KUKA KRL program: EPS_2_25862_MH3A_A_20251016034258.src

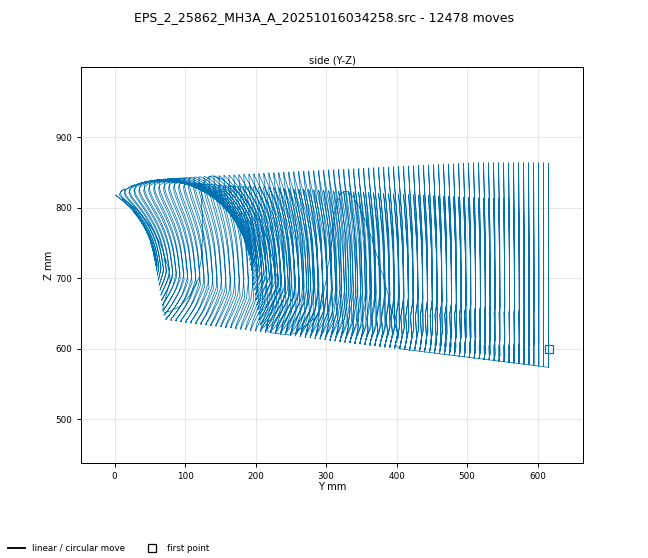
[picture p0: tool path of EPS_2_25862_MH3A_A_20251016034258.src, 12478 of 12480 moves have a stored position in this frame; points joined in program order, loops and branches not executed]
&ACCESS RVP
&REL 4
&COMMENT QRS 19112012
&PARAM EDITMASK = *
DEF PART()
EXT BAS (BAS_COMMAND :IN,REAL :IN )
INT I
BAS (#INITMOV,0 )

;KUKA QRS Post kuka4.cps  Date:22-06-2017 !

File_ID=2889

QRS_PRE_INIT()

;Init var - Until changes are made in qrs_pre_init
Outlet_Square_prg=0
Inlet_1_Square_prg=0
Inlet_2_Square_prg=0
Inlet_3_Square_prg=0
Inlet_4_Square_prg=0
Inlet_5_Square_prg=0

Outlet_1={X 0.000, Y 513.730, Z 763.500, B 0.000, E1 0.000 }
Inlet_1={X 0.000, Y 517.300, Z 713.500, B 0.000, E1 225.000 }
Outlet_1_type=201
Inlet_1_type=201
;QRS#1=Sidecore dimensions
;QRS#2=200-8" PVC SDR 35
;QRS#3=200-8" PVC SDR 35
;QRS#4=
;QRS#5=
;QRS#6=
;QRS#7=
;QRS#8=
;QRS#9=12-08 PSX
;QRS#10=12-08 PSX
;QRS#11=
;QRS#12=
;QRS#13=
;QRS#14=
;QRS#15=
;QRS#16=1220x127x1143 3,75'
;QRS#17=EPS Height
;QRS#18=864
;QRS#19=*
;QRS#20= UPDATED VERSION 22-06-2017
;QRS#21=*
Outlet_Square=0100
Inlet_1_Square=0100
Inlet_2_Square=0
Inlet_3_Square=0
Inlet_4_Square=0
Inlet_5_Square=0
Mill_Square=1
Outlet_Square_Prg=204
Inlet_1_Square_prg=204

QRS_INIT()

$ADVANCE=5

; T1
PTP {E1 173.596,E2 173.596}
PTP {X 0,Y 615.504,A -85,B 0,C 180,E1 173.596,E2 173.596,E3 0,E4 0,E5 0,E6 0}
QRS_SPEED_INIT()
LIN {X 0,Y 615.504,Z 600,A -85,B 0,C 180,E1 173.596,E2 173.596,E3 0,E4 0,E5 0,E6 0} C_VEL
LIN {X 0,Y 615.504,Z 583.862,A -85,B 0,C 180,E1 173.596,E2 173.596} C_VEL
LIN {X 0,Y 615.504,Z 575.681,A -85,B 0,C 180,E1 173.596,E2 173.596} C_VEL
LIN {X 0,Y 615.487,Z 573.681,A -85,B 0,C 180,E1 173.41,E2 173.41} C_VEL
LIN {X 0,Y 615.476,Z 573.691,A -85,B 0,C 180,E1 170.801,E2 170.801} C_VEL
LIN {X 0,Y 615.486,Z 573.696,A -85,B 0,C 180,E1 168.14,E2 168.14} C_VEL
LIN {X 0,Y 615.48,Z 573.683,A -85,B 0,C 180,E1 165.451,E2 165.451} C_VEL
LIN {X 0,Y 615.477,Z 573.689,A -85,B 0,C 180,E1 162.73,E2 162.73} C_VEL
LIN {X 0,Y 615.485,Z 573.695,A -85,B 0,C 180,E1 159.968,E2 159.968} C_VEL
LIN {X 0,Y 615.486,Z 573.681,A -85,B 0,C 180,E1 157.156,E2 157.156} C_VEL
LIN {X 0,Y 615.485,Z 573.696,A -85,B 0,C 180,E1 154.285,E2 154.285} C_VEL
LIN {X 0,Y 615.476,Z 573.69,A -85,B 0,C 180,E1 151.549,E2 151.549} C_VEL
LIN {X 0,Y 615.483,Z 573.682,A -85,B 0,C 180,E1 148.912,E2 148.912} C_VEL
LIN {X 0,Y 615.495,Z 573.699,A -85,B 0,C 180,E1 145.979,E2 145.979} C_VEL
LIN {X 0,Y 615.486,Z 573.682,A -85,B 0,C 180,E1 143.062,E2 143.062} C_VEL
LIN {X 0,Y 615.477,Z 573.691,A -85,B 0,C 180,E1 140.25,E2 140.25} C_VEL
LIN {X 0,Y 615.489,Z 573.697,A -85,B 0,C 180,E1 137.648,E2 137.648} C_VEL
LIN {X 0,Y 615.48,Z 573.684,A -85,B 0,C 180,E1 134.931,E2 134.931} C_VEL
LIN {X 0,Y 615.477,Z 573.691,A -85,B 0,C 180,E1 132.08,E2 132.08} C_VEL
LIN {X 0,Y 615.493,Z 573.697,A -85,B 0,C 180,E1 129.749,E2 129.749} C_VEL
LIN {X 0,Y 615.48,Z 573.685,A -85,B 0,C 180,E1 126.936,E2 126.936} C_VEL
LIN {X 0,Y 615.49,Z 573.681,A -85,B 0,C 180,E1 124.702,E2 124.702} C_VEL
LIN {X 0,Y 615.484,Z 573.682,A -85,B 0,C 180,E1 122.331,E2 122.331} C_VEL
LIN {X 0,Y 615.494,Z 573.7,A -85,B 0,C 180,E1 119.405,E2 119.405} C_VEL
LIN {X 0,Y 615.491,Z 573.68,A -85,B 0,C 180,E1 116.443,E2 116.443} C_VEL
LIN {X 0,Y 615.487,Z 573.695,A -85,B 0,C 180,E1 113.556,E2 113.556} C_VEL
LIN {X 0,Y 615.479,Z 573.687,A -85,B 0,C 180,E1 110.73,E2 110.73} C_VEL
LIN {X 0,Y 615.478,Z 573.685,A -85,B 0,C 180,E1 107.957,E2 107.957} C_VEL
LIN {X 0,Y 615.492,Z 573.701,A -85,B 0,C 180,E1 105.226,E2 105.226} C_VEL
LIN {X 0,Y 615.479,Z 573.686,A -85,B 0,C 180,E1 102.53,E2 102.53} C_VEL
LIN {X 0,Y 615.48,Z 573.684,A -85,B 0,C 180,E1 99.862,E2 99.862} C_VEL
LIN {X 0,Y 615.489,Z 573.696,A -85,B 0,C 180,E1 97.215,E2 97.215} C_VEL
LIN {X 0,Y 615.48,Z 573.69,A -85,B 0,C 180,E1 94.584,E2 94.584} C_VEL
LIN {X 0,Y 615.493,Z 573.68,A -85,B 0,C 180,E1 91.963,E2 91.963} C_VEL
LIN {X 0,Y 615.474,Z 573.691,A -85,B 0,C 180,E1 89.346,E2 89.346} C_VEL
LIN {X 0,Y 615.49,Z 573.697,A -85,B 0,C 180,E1 86.727,E2 86.727} C_VEL
LIN {X 0,Y 615.486,Z 573.683,A -85,B 0,C 180,E1 84.102,E2 84.102} C_VEL
LIN {X 0,Y 615.477,Z 573.685,A -85,B 0,C 180,E1 81.463,E2 81.463} C_VEL
LIN {X 0,Y 615.498,Z 573.697,A -85,B 0,C 180,E1 78.807,E2 78.807} C_VEL
LIN {X 0,Y 615.483,Z 573.686,A -85,B 0,C 180,E1 76.067,E2 76.067} C_VEL
LIN {X 0,Y 615.478,Z 573.684,A -85,B 0,C 180,E1 73.414,E2 73.414} C_VEL
LIN {X 0,Y 615.489,Z 573.699,A -85,B 0,C 180,E1 70.663,E2 70.663} C_VEL
LIN {X 0,Y 615.491,Z 573.681,A -85,B 0,C 180,E1 67.652,E2 67.652} C_VEL
LIN {X 0,Y 615.475,Z 573.688,A -85,B 0,C 180,E1 65.008,E2 65.008} C_VEL
LIN {X 0,Y 615.477,Z 573.878,A -85,B 0,C 180,E1 62.956,E2 62.956} C_VEL
LIN {X 0,Y 615.476,Z 589.581,A -85,B 0,C 180,E1 60.206,E2 60.206} C_VEL
LIN {X 0,Y 615.478,Z 603.411,A -85,B 0,C 180,E1 57.811,E2 57.811} C_VEL
LIN {X 0,Y 615.492,Z 710.1,A -85,B 0,C 180,E1 56.539,E2 56.539} C_VEL
LIN {X 0,Y 615.486,Z 723.119,A -85,B 0,C 180,E1 56.252,E2 56.252} C_VEL
LIN {X 0,Y 615.483,Z 735.365,A -85,B 0,C 180,E1 55.851,E2 55.851} C_VEL
LIN {X 0,Y 615.489,Z 747.801,A -85,B 0,C 180,E1 55.298,E2 55.298} C_VEL
LIN {X 0,Y 615.478,Z 758.469,A -85,B 0,C 180,E1 54.686,E2 54.686} C_VEL
LIN {X 0,Y 615.5,Z 769.773,A -85,B 0,C 180,E1 53.871,E2 53.871} C_VEL
LIN {X 0,Y 615.497,Z 778.829,A -85,B 0,C 180,E1 53.062,E2 53.062} C_VEL
LIN {X 0,Y 615.494,Z 786.885,A -85,B 0,C 180,E1 52.18,E2 52.18} C_VEL
LIN {X 0,Y 615.493,Z 794.893,A -85,B 0,C 180,E1 51.097,E2 51.097} C_VEL
LIN {X 0,Y 615.498,Z 799.899,A -85,B 0,C 180,E1 50.252,E2 50.252} C_VEL
LIN {X 0,Y 615.498,Z 805.113,A -85,B 0,C 180,E1 49.15,E2 49.15} C_VEL
LIN {X 0,Y 615.498,Z 809.309,A -85,B 0,C 180,E1 47.918,E2 47.918} C_VEL
LIN {X 0,Y 615.496,Z 811.875,A -85,B 0,C 180,E1 46.757,E2 46.757} C_VEL
LIN {X 0,Y 615.495,Z 813.002,A -85,B 0,C 180,E1 45.853,E2 45.853} C_VEL
LIN {X 0,Y 615.495,Z 813.388,A -85,B 0,C 180,E1 44.934,E2 44.934} C_VEL
LIN {X 0,Y 615.493,Z 812.962,A -85,B 0,C 180,E1 44,E2 44} C_VEL
LIN {X 0,Y 615.497,Z 811.704,A -85,B 0,C 180,E1 43.05,E2 43.05} C_VEL
LIN {X 0,Y 615.496,Z 809.552,A -85,B 0,C 180,E1 42.083,E2 42.083} C_VEL
LIN {X 0,Y 615.493,Z 806.404,A -85,B 0,C 180,E1 41.097,E2 41.097} C_VEL
LIN {X 0,Y 615.497,Z 802.114,A -85,B 0,C 180,E1 40.092,E2 40.092} C_VEL
LIN {X 0,Y 615.497,Z 796.474,A -85,B 0,C 180,E1 39.065,E2 39.065} C_VEL
LIN {X 0,Y 615.495,Z 789.205,A -85,B 0,C 180,E1 38.015,E2 38.015} C_VEL
LIN {X 0,Y 615.498,Z 781.195,A -85,B 0,C 180,E1 37.09,E2 37.09} C_VEL
LIN {X 0,Y 615.499,Z 772.601,A -85,B 0,C 180,E1 36.276,E2 36.276} C_VEL
LIN {X 0,Y 615.495,Z 762.802,A -85,B 0,C 180,E1 35.514,E2 35.514} C_VEL
LIN {X 0,Y 615.483,Z 751.624,A -85,B 0,C 180,E1 34.815,E2 34.815} C_VEL
LIN {X 0,Y 615.489,Z 739.667,A -85,B 0,C 180,E1 34.233,E2 34.233} C_VEL
LIN {X 0,Y 615.48,Z 727.257,A -85,B 0,C 180,E1 33.778,E2 33.778} C_VEL
LIN {X 0,Y 615.474,Z 714.959,A -85,B 0,C 180,E1 33.46,E2 33.46} C_VEL
LIN {X 0,Y 615.48,Z 700.03,A -85,B 0,C 180,E1 33.236,E2 33.236} C_VEL
LIN {X 0,Y 615.483,Z 603.35,A -85,B 0,C 180,E1 32.089,E2 32.089} C_VEL
LIN {X 0,Y 615.49,Z 586.786,A -85,B 0,C 180,E1 29.218,E2 29.218} C_VEL
LIN {X 0,Y 615.496,Z 573.683,A -85,B 0,C 180,E1 26.897,E2 26.897} C_VEL
LIN {X 0,Y 615.485,Z 573.686,A -85,B 0,C 180,E1 24.011,E2 24.011} C_VEL
LIN {X 0,Y 615.495,Z 573.7,A -85,B 0,C 180,E1 21.431,E2 21.431} C_VEL
LIN {X 0,Y 615.483,Z 573.683,A -85,B 0,C 180,E1 18.608,E2 18.608} C_VEL
LIN {X 0,Y 615.483,Z 573.686,A -85,B 0,C 180,E1 15.905,E2 15.905} C_VEL
LIN {X 0,Y 615.495,Z 573.697,A -85,B 0,C 180,E1 13.201,E2 13.201} C_VEL
LIN {X 0,Y 615.485,Z 573.683,A -85,B 0,C 180,E1 10.527,E2 10.527} C_VEL
LIN {X 0,Y 615.482,Z 573.685,A -85,B 0,C 180,E1 7.875,E2 7.875} C_VEL
LIN {X 0,Y 615.487,Z 573.701,A -85,B 0,C 180,E1 5.241,E2 5.241} C_VEL
LIN {X 0,Y 615.496,Z 573.684,A -85,B 0,C 180,E1 2.617,E2 2.617} C_VEL
LIN {X 0,Y 615.476,Z 573.684,A -85,B 0,C 180,E1 0,E2 0} C_VEL
LIN {X 0,Y 615.496,Z 573.69,A -85,B 0,C 180,E1 -2.618,E2 -2.618} C_VEL
LIN {X 0,Y 615.49,Z 573.691,A -85,B 0,C 180,E1 -5.242,E2 -5.242} C_VEL
LIN {X 0,Y 615.482,Z 573.683,A -85,B 0,C 180,E1 -7.876,E2 -7.876} C_VEL
LIN {X 0,Y 615.484,Z 573.688,A -85,B 0,C 180,E1 -10.527,E2 -10.527} C_VEL
LIN {X 0,Y 615.49,Z 573.696,A -85,B 0,C 180,E1 -13.201,E2 -13.201} C_VEL
LIN {X 0,Y 615.483,Z 573.683,A -85,B 0,C 180,E1 -15.906,E2 -15.906} C_VEL
LIN {X 0,Y 615.484,Z 573.688,A -85,B 0,C 180,E1 -18.646,E2 -18.646} C_VEL
LIN {X 0,Y 615.486,Z 573.693,A -85,B 0,C 180,E1 -21.432,E2 -21.432} C_VEL
LIN {X 0,Y 615.478,Z 573.684,A -85,B 0,C 180,E1 -24.273,E2 -24.273} C_VEL
LIN {X 0,Y 615.492,Z 573.695,A -85,B 0,C 180,E1 -27.049,E2 -27.049} C_VEL
LIN {X 0,Y 615.49,Z 573.685,A -85,B 0,C 180,E1 -29.797,E2 -29.797} C_VEL
LIN {X 0,Y 615.477,Z 573.684,A -85,B 0,C 180,E1 -32.458,E2 -32.458} C_VEL
LIN {X 0,Y 615.477,Z 573.689,A -85,B 0,C 180,E1 -34.816,E2 -34.816} C_VEL
LIN {X 0,Y 615.492,Z 573.697,A -85,B 0,C 180,E1 -37.242,E2 -37.242} C_VEL
LIN {X 0,Y 615.495,Z 573.682,A -85,B 0,C 180,E1 -40.092,E2 -40.092} C_VEL
LIN {X 0,Y 615.488,Z 573.681,A -85,B 0,C 180,E1 -42.353,E2 -42.353} C_VEL
LIN {X 0,Y 615.481,Z 573.691,A -85,B 0,C 180,E1 -45.07,E2 -45.07} C_VEL
LIN {X 0,Y 615.483,Z 573.69,A -85,B 0,C 180,E1 -47.921,E2 -47.921} C_VEL
LIN {X 0,Y 615.494,Z 573.681,A -85,B 0,C 180,E1 -50.252,E2 -50.252} C_VEL
LIN {X 0,Y 615.478,Z 573.689,A -85,B 0,C 180,E1 -53.065,E2 -53.065} C_VEL
LIN {X 0,Y 615.49,Z 573.691,A -85,B 0,C 180,E1 -55.3,E2 -55.3} C_VEL
LIN {X 0,Y 615.494,Z 573.7,A -85,B 0,C 180,E1 -57.669,E2 -57.669} C_VEL
LIN {X 0,Y 615.493,Z 573.68,A -85,B 0,C 180,E1 -60.595,E2 -60.595} C_VEL
LIN {X 0,Y 615.491,Z 573.696,A -85,B 0,C 180,E1 -63.557,E2 -63.557} C_VEL
LIN {X 0,Y 615.489,Z 573.683,A -85,B 0,C 180,E1 -66.444,E2 -66.444} C_VEL
LIN {X 0,Y 615.475,Z 573.827,A -85,B 0,C 180,E1 -67.067,E2 -67.067} C_VEL
LIN {X 0,Y 615.486,Z 594.759,A -85,B 0,C 180,E1 -69.837,E2 -69.837} C_VEL
LIN {X 0,Y 615.497,Z 616.999,A -85,B 0,C 180,E1 -72.73,E2 -72.73} C_VEL
LIN {X 0,Y 615.484,Z 639.434,A -85,B 0,C 180,E1 -75.606,E2 -75.606} C_VEL
LIN {X 0,Y 615.478,Z 651.3,A -85,B 0,C 180,E1 -77.114,E2 -77.114} C_VEL
LIN {X 0,Y 615.477,Z 759.849,A -85,B 0,C 180,E1 -78.411,E2 -78.411} C_VEL
LIN {X 0,Y 615.488,Z 772.354,A -85,B 0,C 180,E1 -78.682,E2 -78.682} C_VEL
LIN {X 0,Y 615.496,Z 785.512,A -85,B 0,C 180,E1 -79.109,E2 -79.109} C_VEL
LIN {X 0,Y 615.484,Z 797.482,A -85,B 0,C 180,E1 -79.64,E2 -79.64} C_VEL
LIN {X 0,Y 615.483,Z 809,A -85,B 0,C 180,E1 -80.304,E2 -80.304} C_VEL
LIN {X 0,Y 615.499,Z 819.344,A -85,B 0,C 180,E1 -81.05,E2 -81.05} C_VEL
LIN {X 0,Y 615.497,Z 827.814,A -85,B 0,C 180,E1 -81.794,E2 -81.794} C_VEL
LIN {X 0,Y 615.498,Z 835.608,A -85,B 0,C 180,E1 -82.62,E2 -82.62} C_VEL
LIN {X 0,Y 615.496,Z 843.204,A -85,B 0,C 180,E1 -83.608,E2 -83.608} C_VEL
LIN {X 0,Y 615.498,Z 850.205,A -85,B 0,C 180,E1 -84.759,E2 -84.759} C_VEL
LIN {X 0,Y 615.494,Z 854.852,A -85,B 0,C 180,E1 -85.744,E2 -85.744} C_VEL
LIN {X 0,Y 615.496,Z 858.399,A -85,B 0,C 180,E1 -86.727,E2 -86.727} C_VEL
LIN {X 0,Y 615.497,Z 860.233,A -85,B 0,C 180,E1 -87.382,E2 -87.382} C_VEL
LIN {X 0,Y 615.496,Z 861.608,A -85,B 0,C 180,E1 -88.037,E2 -88.037} C_VEL
LIN {X 0,Y 615.496,Z 863.174,A -85,B 0,C 180,E1 -89.346,E2 -89.346} C_VEL
LIN {X 0,Y 615.494,Z 863.389,A -85,B 0,C 180,E1 -90,E2 -90} C_VEL
LIN {X 0,Y 615.496,Z 862.58,A -85,B 0,C 180,E1 -91.309,E2 -91.309} C_VEL
LIN {X 0,Y 615.496,Z 861.608,A -85,B 0,C 180,E1 -91.963,E2 -91.963} C_VEL
LIN {X 0,Y 615.497,Z 860.233,A -85,B 0,C 180,E1 -92.618,E2 -92.618} C_VEL
LIN {X 0,Y 615.496,Z 857.35,A -85,B 0,C 180,E1 -93.601,E2 -93.601} C_VEL
LIN {X 0,Y 615.498,Z 853.442,A -85,B 0,C 180,E1 -94.584,E2 -94.584} C_VEL
LIN {X 0,Y 615.499,Z 848.406,A -85,B 0,C 180,E1 -95.57,E2 -95.57} C_VEL
LIN {X 0,Y 615.497,Z 841.87,A -85,B 0,C 180,E1 -96.583,E2 -96.583} C_VEL
LIN {X 0,Y 615.497,Z 834.135,A -85,B 0,C 180,E1 -97.545,E2 -97.545} C_VEL
LIN {X 0,Y 615.498,Z 826.047,A -85,B 0,C 180,E1 -98.371,E2 -98.371} C_VEL
LIN {X 0,Y 615.499,Z 816.17,A -85,B 0,C 180,E1 -99.198,E2 -99.198} C_VEL
LIN {X 0,Y 615.487,Z 804.986,A -85,B 0,C 180,E1 -99.945,E2 -99.945} C_VEL
LIN {X 0,Y 615.483,Z 794.029,A -85,B 0,C 180,E1 -100.527,E2 -100.527} C_VEL
LIN {X 0,Y 615.496,Z 781.436,A -85,B 0,C 180,E1 -101.042,E2 -101.042} C_VEL
LIN {X 0,Y 615.483,Z 769.078,A -85,B 0,C 180,E1 -101.401,E2 -101.401} C_VEL
LIN {X 0,Y 615.477,Z 755.49,A -85,B 0,C 180,E1 -101.652,E2 -101.652} C_VEL
LIN {X 0,Y 615.478,Z 651.3,A -85,B 0,C 180,E1 -102.886,E2 -102.886} C_VEL
LIN {X 0,Y 615.48,Z 630.263,A -85,B 0,C 180,E1 -105.565,E2 -105.565} C_VEL
LIN {X 0,Y 615.498,Z 609.208,A -85,B 0,C 180,E1 -108.278,E2 -108.278} C_VEL
LIN {X 0,Y 615.489,Z 586.457,A -85,B 0,C 180,E1 -111.256,E2 -111.256} C_VEL
LIN {X 0,Y 615.477,Z 573.685,A -85,B 0,C 180,E1 -112.978,E2 -112.978} C_VEL
LIN {X 0,Y 615.484,Z 573.686,A -85,B 0,C 180,E1 -115.715,E2 -115.715} C_VEL
LIN {X 0,Y 615.494,Z 573.697,A -85,B 0,C 180,E1 -118.451,E2 -118.451} C_VEL
LIN {X 0,Y 615.473,Z 573.686,A -85,B 0,C 180,E1 -121.083,E2 -121.083} C_VEL
LIN {X 0,Y 615.495,Z 573.679,A -85,B 0,C 180,E1 -123.535,E2 -123.535} C_VEL
LIN {X 0,Y 615.487,Z 573.7,A -85,B 0,C 180,E1 -126.424,E2 -126.424} C_VEL
LIN {X 0,Y 615.476,Z 573.689,A -85,B 0,C 180,E1 -129.06,E2 -129.06} C_VEL
LIN {X 0,Y 615.481,Z 573.683,A -85,B 0,C 180,E1 -131.473,E2 -131.473} C_VEL
LIN {X 0,Y 615.481,Z 573.688,A -85,B 0,C 180,E1 -134.149,E2 -134.149} C_VEL
LIN {X 0,Y 615.484,Z 573.693,A -85,B 0,C 180,E1 -136.951,E2 -136.951} C_VEL
LIN {X 0,Y 615.473,Z 573.687,A -85,B 0,C 180,E1 -139.392,E2 -139.392} C_VEL
LIN {X 0,Y 615.486,Z 573.682,A -85,B 0,C 180,E1 -141.986,E2 -141.986} C_VEL
LIN {X 0,Y 615.48,Z 573.69,A -85,B 0,C 180,E1 -144.383,E2 -144.383} C_VEL
LIN {X 0,Y 615.486,Z 573.699,A -85,B 0,C 180,E1 -146.763,E2 -146.763} C_VEL
LIN {X 0,Y 615.487,Z 573.696,A -85,B 0,C 180,E1 -149.08,E2 -149.08} C_VEL
LIN {X 0,Y 615.476,Z 573.687,A -85,B 0,C 180,E1 -151.549,E2 -151.549} C_VEL
LIN {X 0,Y 615.486,Z 573.683,A -85,B 0,C 180,E1 -154.284,E2 -154.284} C_VEL
LIN {X 0,Y 615.488,Z 573.698,A -85,B 0,C 180,E1 -157.155,E2 -157.155} C_VEL
LIN {X 0,Y 615.485,Z 573.682,A -85,B 0,C 180,E1 -159.967,E2 -159.967} C_VEL
LIN {X 0,Y 615.479,Z 573.69,A -85,B 0,C 180,E1 -162.729,E2 -162.729} C_VEL
LIN {X 0,Y 615.48,Z 573.695,A -85,B 0,C 180,E1 -165.45,E2 -165.45} C_VEL
LIN {X 0,Y 615.485,Z 573.682,A -85,B 0,C 180,E1 -168.139,E2 -168.139} C_VEL
LIN {X 0,Y 615.478,Z 573.689,A -85,B 0,C 180,E1 -170.801,E2 -170.801} C_VEL
LIN {X 0,Y 615.489,Z 573.698,A -85,B 0,C 180,E1 -173.443,E2 -173.443} C_VEL
LIN {X 0,Y 615.477,Z 573.685,A -85,B 0,C 180,E1 -176.071,E2 -176.071} C_VEL
LIN {X 0,Y 615.485,Z 573.683,A -85,B 0,C 180,E1 -178.691,E2 -178.691} C_VEL
LIN {X 0,Y 615.487,Z 573.696,A -85,B 0,C 180,E1 -181.308,E2 -181.308} C_VEL
LIN {X 0,Y 615.477,Z 573.691,A -85,B 0,C 180,E1 -183.928,E2 -183.928} C_VEL
LIN {X 0,Y 615.487,Z 573.681,A -85,B 0,C 180,E1 -186.59,E2 -186.59} C_VEL
LIN {X 0,Y 614.805,Z 573.839,A -85,B 0,C 180,E1 -187.136,E2 -187.136} C_VEL
LIN {X 0,Y 611.964,Z 574.253,A -85,B 0,C 180,E1 -188.022,E2 -188.022} C_VEL
LIN {X 0,Y 609.571,Z 574.564,A -85,B 0,C 180,E1 -188.735,E2 -188.735} C_VEL
LIN {X 0,Y 608.539,Z 574.682,A -85,B 0,C 180,E1 -189.284,E2 -189.284} C_VEL
LIN {X 0,Y 608.452,Z 574.691,A -85,B 0,C 180,E1 -189.47,E2 -189.47} C_VEL
LIN {X 0,Y 608.46,Z 574.691,A -85,B 0,C 180,E1 -191.999,E2 -191.999} C_VEL
LIN {X 0,Y 608.467,Z 574.685,A -85,B 0,C 180,E1 -194.72,E2 -194.72} C_VEL
LIN {X 0,Y 608.446,Z 574.693,A -85,B 0,C 180,E1 -197.476,E2 -197.476} C_VEL
LIN {X 0,Y 608.459,Z 574.689,A -85,B 0,C 180,E1 -200.274,E2 -200.274} C_VEL
LIN {X 0,Y 608.447,Z 574.688,A -85,B 0,C 180,E1 -203.124,E2 -203.124} C_VEL
LIN {X 0,Y 608.466,Z 574.693,A -85,B 0,C 180,E1 -205.723,E2 -205.723} C_VEL
LIN {X 0,Y 608.444,Z 574.693,A -85,B 0,C 180,E1 -208.267,E2 -208.267} C_VEL
LIN {X 0,Y 608.47,Z 574.687,A -85,B 0,C 180,E1 -210.544,E2 -210.544} C_VEL
LIN {X 0,Y 608.45,Z 574.687,A -85,B 0,C 180,E1 -212.879,E2 -212.879} C_VEL
LIN {X 0,Y 608.434,Z 574.689,A -85,B 0,C 180,E1 -215.278,E2 -215.278} C_VEL
LIN {X 0,Y 608.471,Z 574.689,A -85,B 0,C 180,E1 -217.746,E2 -217.746} C_VEL
LIN {X 0,Y 608.472,Z 574.693,A -85,B 0,C 180,E1 -220.333,E2 -220.333} C_VEL
LIN {X 0,Y 608.483,Z 574.683,A -85,B 0,C 180,E1 -223.312,E2 -223.312} C_VEL
LIN {X 0,Y 608.465,Z 574.693,A -85,B 0,C 180,E1 -226.132,E2 -226.132} C_VEL
LIN {X 0,Y 608.447,Z 574.69,A -85,B 0,C 180,E1 -228.824,E2 -228.824} C_VEL
LIN {X 0,Y 608.462,Z 574.685,A -85,B 0,C 180,E1 -231.413,E2 -231.413} C_VEL
LIN {X 0,Y 608.471,Z 574.687,A -85,B 0,C 180,E1 -233.951,E2 -233.951} C_VEL
LIN {X 0,Y 608.467,Z 574.694,A -85,B 0,C 180,E1 -236.33,E2 -236.33} C_VEL
LIN {X 0,Y 608.471,Z 574.692,A -85,B 0,C 180,E1 -238.728,E2 -238.728} C_VEL
LIN {X 0,Y 608.473,Z 574.684,A -85,B 0,C 180,E1 -241.379,E2 -241.379} C_VEL
LIN {X 0,Y 608.443,Z 574.689,A -85,B 0,C 180,E1 -243.965,E2 -243.965} C_VEL
LIN {X 0,Y 608.461,Z 574.688,A -85,B 0,C 180,E1 -246.156,E2 -246.156} C_VEL
LIN {X 0,Y 608.47,Z 574.689,A -85,B 0,C 180,E1 -248.309,E2 -248.309} C_VEL
LIN {X 0,Y 608.465,Z 574.688,A -85,B 0,C 180,E1 -251.284,E2 -251.284} C_VEL
LIN {X 0,Y 608.456,Z 574.686,A -85,B 0,C 180,E1 -253.906,E2 -253.906} C_VEL
LIN {X 0,Y 608.469,Z 574.692,A -85,B 0,C 180,E1 -256.644,E2 -256.644} C_VEL
LIN {X 0,Y 608.459,Z 574.689,A -85,B 0,C 180,E1 -259.35,E2 -259.35} C_VEL
LIN {X 0,Y 608.473,Z 574.684,A -85,B 0,C 180,E1 -262.033,E2 -262.033} C_VEL
LIN {X 0,Y 608.465,Z 574.691,A -85,B 0,C 180,E1 -264.698,E2 -264.698} C_VEL
LIN {X 0,Y 608.472,Z 574.69,A -85,B 0,C 180,E1 -267.352,E2 -267.352} C_VEL
LIN {X 0,Y 608.477,Z 574.684,A -85,B 0,C 180,E1 -270,E2 -270} C_VEL
LIN {X 0,Y 608.469,Z 574.688,A -85,B 0,C 180,E1 -272.648,E2 -272.648} C_VEL
LIN {X 0,Y 608.469,Z 574.694,A -85,B 0,C 180,E1 -275.302,E2 -275.302} C_VEL
LIN {X 0,Y 608.475,Z 574.685,A -85,B 0,C 180,E1 -277.967,E2 -277.967} C_VEL
LIN {X 0,Y 608.456,Z 574.688,A -85,B 0,C 180,E1 -280.65,E2 -280.65} C_VEL
LIN {X 0,Y 608.47,Z 574.695,A -85,B 0,C 180,E1 -283.356,E2 -283.356} C_VEL
LIN {X 0,Y 608.458,Z 574.687,A -85,B 0,C 180,E1 -286.093,E2 -286.093} C_VEL
LIN {X 0,Y 608.451,Z 574.689,A -85,B 0,C 180,E1 -288.869,E2 -288.869} C_VEL
LIN {X 0,Y 608.472,Z 574.691,A -85,B 0,C 180,E1 -291.691,E2 -291.691} C_VEL
LIN {X 0,Y 608.451,Z 574.687,A -85,B 0,C 180,E1 -294.571,E2 -294.571} C_VEL
LIN {X 0,Y 608.46,Z 574.713,A -85,B 0,C 180,E1 -296.963,E2 -296.963} C_VEL
LIN {X 0,Y 608.48,Z 589.567,A -85,B 0,C 180,E1 -299.588,E2 -299.588} C_VEL
LIN {X 0,Y 608.442,Z 603.672,A -85,B 0,C 180,E1 -302.046,E2 -302.046} C_VEL
LIN {X 0,Y 608.562,Z 710.327,A -85,B 0,C 180,E1 -303.329,E2 -303.329} C_VEL
LIN {X 0,Y 608.528,Z 723.641,A -85,B 0,C 180,E1 -303.628,E2 -303.628} C_VEL
LIN {X 0,Y 608.521,Z 736.649,A -85,B 0,C 180,E1 -304.066,E2 -304.066} C_VEL
LIN {X 0,Y 608.493,Z 749.042,A -85,B 0,C 180,E1 -304.639,E2 -304.639} C_VEL
LIN {X 0,Y 608.473,Z 759.786,A -85,B 0,C 180,E1 -305.275,E2 -305.275} C_VEL
LIN {X 0,Y 608.48,Z 770.82,A -85,B 0,C 180,E1 -306.089,E2 -306.089} C_VEL
LIN {X 0,Y 608.459,Z 781.01,A -85,B 0,C 180,E1 -307.036,E2 -307.036} C_VEL
LIN {X 0,Y 608.452,Z 789.332,A -85,B 0,C 180,E1 -307.991,E2 -307.991} C_VEL
LIN {X 0,Y 608.437,Z 797.122,A -85,B 0,C 180,E1 -309.12,E2 -309.12} C_VEL
LIN {X 0,Y 608.443,Z 803.471,A -85,B 0,C 180,E1 -310.303,E2 -310.303} C_VEL
LIN {X 0,Y 608.427,Z 807.675,A -85,B 0,C 180,E1 -311.339,E2 -311.339} C_VEL
LIN {X 0,Y 608.437,Z 810.639,A -85,B 0,C 180,E1 -312.332,E2 -312.332} C_VEL
LIN {X 0,Y 608.432,Z 812.611,A -85,B 0,C 180,E1 -313.306,E2 -313.306} C_VEL
LIN {X 0,Y 608.418,Z 813.697,A -85,B 0,C 180,E1 -314.261,E2 -314.261} C_VEL
LIN {X 0,Y 608.417,Z 813.969,A -85,B 0,C 180,E1 -315.201,E2 -315.201} C_VEL
LIN {X 0,Y 608.427,Z 813.468,A -85,B 0,C 180,E1 -316.127,E2 -316.127} C_VEL
LIN {X 0,Y 608.435,Z 812.188,A -85,B 0,C 180,E1 -317.039,E2 -317.039} C_VEL
LIN {X 0,Y 608.425,Z 810.162,A -85,B 0,C 180,E1 -317.936,E2 -317.936} C_VEL
LIN {X 0,Y 608.43,Z 807.411,A -85,B 0,C 180,E1 -318.822,E2 -318.822} C_VEL
LIN {X 0,Y 608.444,Z 802.859,A -85,B 0,C 180,E1 -319.913,E2 -319.913} C_VEL
LIN {X 0,Y 608.437,Z 796.597,A -85,B 0,C 180,E1 -321.057,E2 -321.057} C_VEL
LIN {X 0,Y 608.453,Z 790.022,A -85,B 0,C 180,E1 -322.008,E2 -322.008} C_VEL
LIN {X 0,Y 608.46,Z 781.895,A -85,B 0,C 180,E1 -322.963,E2 -322.963} C_VEL
LIN {X 0,Y 608.477,Z 771.877,A -85,B 0,C 180,E1 -323.91,E2 -323.91} C_VEL
LIN {X 0,Y 608.486,Z 761.147,A -85,B 0,C 180,E1 -324.726,E2 -324.726} C_VEL
LIN {X 0,Y 608.488,Z 749.127,A -85,B 0,C 180,E1 -325.446,E2 -325.446} C_VEL
LIN {X 0,Y 608.534,Z 737.604,A -85,B 0,C 180,E1 -325.985,E2 -325.985} C_VEL
LIN {X 0,Y 608.512,Z 724.711,A -85,B 0,C 180,E1 -326.432,E2 -326.432} C_VEL
LIN {X 0,Y 608.531,Z 711.345,A -85,B 0,C 180,E1 -326.743,E2 -326.743} C_VEL
LIN {X 0,Y 608.555,Z 678.685,A -85,B 0,C 180,E1 -327.153,E2 -327.153} C_VEL
LIN {X 0,Y 608.474,Z 603.606,A -85,B 0,C 180,E1 -328.053,E2 -328.053} C_VEL
LIN {X 0,Y 608.487,Z 586.839,A -85,B 0,C 180,E1 -330.982,E2 -330.982} C_VEL
LIN {X 0,Y 608.48,Z 574.686,A -85,B 0,C 180,E1 -333.151,E2 -333.151} C_VEL
LIN {X 0,Y 608.466,Z 574.689,A -85,B 0,C 180,E1 -336.156,E2 -336.156} C_VEL
LIN {X 0,Y 608.458,Z 574.69,A -85,B 0,C 180,E1 -339.019,E2 -339.019} C_VEL
LIN {X 0,Y 608.449,Z 574.688,A -85,B 0,C 180,E1 -341.829,E2 -341.829} C_VEL
LIN {X 0,Y 608.472,Z 574.694,A -85,B 0,C 180,E1 -344.594,E2 -344.594} C_VEL
LIN {X 0,Y 608.476,Z 574.686,A -85,B 0,C 180,E1 -347.323,E2 -347.323} C_VEL
LIN {X 0,Y 608.454,Z 574.687,A -85,B 0,C 180,E1 -350.023,E2 -350.023} C_VEL
LIN {X 0,Y 608.48,Z 574.693,A -85,B 0,C 180,E1 -352.701,E2 -352.701} C_VEL
LIN {X 0,Y 608.467,Z 574.687,A -85,B 0,C 180,E1 -355.363,E2 -355.363} C_VEL
LIN {X 0,Y 608.447,Z 574.688,A -85,B 0,C 180,E1 -358.015,E2 -358.015} C_VEL
LIN {X 0,Y 608.48,Z 574.69,A -85,B 0,C 180,E1 -360.662,E2 -360.662} C_VEL
LIN {X 0,Y 608.479,Z 574.688,A -85,B 0,C 180,E1 -363.311,E2 -363.311} C_VEL
LIN {X 0,Y 608.476,Z 574.684,A -85,B 0,C 180,E1 -365.967,E2 -365.967} C_VEL
LIN {X 0,Y 608.46,Z 574.691,A -85,B 0,C 180,E1 -368.636,E2 -368.636} C_VEL
LIN {X 0,Y 608.476,Z 574.69,A -85,B 0,C 180,E1 -371.324,E2 -371.324} C_VEL
LIN {X 0,Y 608.458,Z 574.686,A -85,B 0,C 180,E1 -374.038,E2 -374.038} C_VEL
LIN {X 0,Y 608.472,Z 574.69,A -85,B 0,C 180,E1 -376.784,E2 -376.784} C_VEL
LIN {X 0,Y 608.453,Z 574.69,A -85,B 0,C 180,E1 -379.571,E2 -379.571} C_VEL
LIN {X 0,Y 608.466,Z 574.686,A -85,B 0,C 180,E1 -382.406,E2 -382.406} C_VEL
LIN {X 0,Y 608.449,Z 574.689,A -85,B 0,C 180,E1 -384.572,E2 -384.572} C_VEL
LIN {X 0,Y 608.481,Z 574.694,A -85,B 0,C 180,E1 -387.21,E2 -387.21} C_VEL
LIN {X 0,Y 608.469,Z 574.686,A -85,B 0,C 180,E1 -389.974,E2 -389.974} C_VEL
LIN {X 0,Y 608.452,Z 574.687,A -85,B 0,C 180,E1 -392.523,E2 -392.523} C_VEL
LIN {X 0,Y 608.469,Z 574.688,A -85,B 0,C 180,E1 -394.91,E2 -394.91} C_VEL
LIN {X 0,Y 608.473,Z 574.689,A -85,B 0,C 180,E1 -397.746,E2 -397.746} C_VEL
LIN {X 0,Y 608.451,Z 574.687,A -85,B 0,C 180,E1 -400.331,E2 -400.331} C_VEL
LIN {X 0,Y 608.451,Z 574.69,A -85,B 0,C 180,E1 -402.96,E2 -402.96} C_VEL
LIN {X 0,Y 608.453,Z 574.693,A -85,B 0,C 180,E1 -405.737,E2 -405.737} C_VEL
LIN {X 0,Y 608.455,Z 574.687,A -85,B 0,C 180,E1 -408.659,E2 -408.659} C_VEL
LIN {X 0,Y 608.465,Z 574.694,A -85,B 0,C 180,E1 -411.413,E2 -411.413} C_VEL
LIN {X 0,Y 608.477,Z 574.688,A -85,B 0,C 180,E1 -413.951,E2 -413.951} C_VEL
LIN {X 0,Y 608.468,Z 574.686,A -85,B 0,C 180,E1 -416.331,E2 -416.331} C_VEL
LIN {X 0,Y 608.443,Z 574.688,A -85,B 0,C 180,E1 -418.733,E2 -418.733} C_VEL
LIN {X 0,Y 608.473,Z 574.69,A -85,B 0,C 180,E1 -421.381,E2 -421.381} C_VEL
LIN {X 0,Y 608.469,Z 574.687,A -85,B 0,C 180,E1 -424.28,E2 -424.28} C_VEL
LIN {X 0,Y 608.476,Z 574.825,A -85,B 0,C 180,E1 -426.923,E2 -426.923} C_VEL
LIN {X 0,Y 608.586,Z 590.447,A -85,B 0,C 180,E1 -429.024,E2 -429.024} C_VEL
LIN {X 0,Y 608.527,Z 611.72,A -85,B 0,C 180,E1 -431.831,E2 -431.831} C_VEL
LIN {X 0,Y 608.491,Z 632.993,A -85,B 0,C 180,E1 -434.595,E2 -434.595} C_VEL
LIN {X 0,Y 608.478,Z 651.524,A -85,B 0,C 180,E1 -436.973,E2 -436.973} C_VEL
LIN {X 0,Y 608.533,Z 759.963,A -85,B 0,C 180,E1 -438.277,E2 -438.277} C_VEL
LIN {X 0,Y 608.536,Z 773.227,A -85,B 0,C 180,E1 -438.572,E2 -438.572} C_VEL
LIN {X 0,Y 608.544,Z 786.343,A -85,B 0,C 180,E1 -439.01,E2 -439.01} C_VEL
LIN {X 0,Y 608.501,Z 797.64,A -85,B 0,C 180,E1 -439.519,E2 -439.519} C_VEL
LIN {X 0,Y 608.474,Z 809.201,A -85,B 0,C 180,E1 -440.191,E2 -440.191} C_VEL
LIN {X 0,Y 608.485,Z 819.596,A -85,B 0,C 180,E1 -440.946,E2 -440.946} C_VEL
LIN {X 0,Y 608.475,Z 828.114,A -85,B 0,C 180,E1 -441.699,E2 -441.699} C_VEL
LIN {X 0,Y 608.471,Z 835.962,A -85,B 0,C 180,E1 -442.534,E2 -442.534} C_VEL
LIN {X 0,Y 608.461,Z 843.287,A -85,B 0,C 180,E1 -443.485,E2 -443.485} C_VEL
LIN {X 0,Y 608.45,Z 848.867,A -85,B 0,C 180,E1 -444.366,E2 -444.366} C_VEL
LIN {X 0,Y 608.432,Z 853.951,A -85,B 0,C 180,E1 -445.362,E2 -445.362} C_VEL
LIN {X 0,Y 608.449,Z 857.896,A -85,B 0,C 180,E1 -446.358,E2 -446.358} C_VEL
LIN {X 0,Y 608.425,Z 860.809,A -85,B 0,C 180,E1 -447.352,E2 -447.352} C_VEL
LIN {X 0,Y 608.441,Z 862.201,A -85,B 0,C 180,E1 -448.014,E2 -448.014} C_VEL
LIN {X 0,Y 608.438,Z 863.783,A -85,B 0,C 180,E1 -449.338,E2 -449.338} C_VEL
LIN {X 0,Y 608.434,Z 864,A -85,B 0,C 180,E1 -450,E2 -450} C_VEL
LIN {X 0,Y 608.448,Z 863.184,A -85,B 0,C 180,E1 -451.324,E2 -451.324} C_VEL
LIN {X 0,Y 608.441,Z 862.201,A -85,B 0,C 180,E1 -451.986,E2 -451.986} C_VEL
LIN {X 0,Y 608.425,Z 860.809,A -85,B 0,C 180,E1 -452.648,E2 -452.648} C_VEL
LIN {X 0,Y 608.449,Z 857.896,A -85,B 0,C 180,E1 -453.642,E2 -453.642} C_VEL
LIN {X 0,Y 608.432,Z 853.951,A -85,B 0,C 180,E1 -454.638,E2 -454.638} C_VEL
LIN {X 0,Y 608.437,Z 847.877,A -85,B 0,C 180,E1 -455.801,E2 -455.801} C_VEL
LIN {X 0,Y 608.462,Z 841.236,A -85,B 0,C 180,E1 -456.799,E2 -456.799} C_VEL
LIN {X 0,Y 608.456,Z 832.991,A -85,B 0,C 180,E1 -457.8,E2 -457.8} C_VEL
LIN {X 0,Y 608.472,Z 824.539,A -85,B 0,C 180,E1 -458.636,E2 -458.636} C_VEL
LIN {X 0,Y 608.471,Z 814.094,A -85,B 0,C 180,E1 -459.473,E2 -459.473} C_VEL
LIN {X 0,Y 608.487,Z 803.76,A -85,B 0,C 180,E1 -460.145,E2 -460.145} C_VEL
LIN {X 0,Y 608.521,Z 792.25,A -85,B 0,C 180,E1 -460.741,E2 -460.741} C_VEL
LIN {X 0,Y 608.538,Z 779.887,A -85,B 0,C 180,E1 -461.225,E2 -461.225} C_VEL
LIN {X 0,Y 608.535,Z 766.451,A -85,B 0,C 180,E1 -461.597,E2 -461.597} C_VEL
LIN {X 0,Y 608.541,Z 754.107,A -85,B 0,C 180,E1 -461.808,E2 -461.808} C_VEL
LIN {X 0,Y 608.467,Z 651.441,A -85,B 0,C 180,E1 -463.037,E2 -463.037} C_VEL
LIN {X 0,Y 608.485,Z 630.334,A -85,B 0,C 180,E1 -465.749,E2 -465.749} C_VEL
LIN {X 0,Y 608.548,Z 609.232,A -85,B 0,C 180,E1 -468.494,E2 -468.494} C_VEL
LIN {X 0,Y 608.568,Z 587.788,A -85,B 0,C 180,E1 -471.332,E2 -471.332} C_VEL
LIN {X 0,Y 608.468,Z 574.687,A -85,B 0,C 180,E1 -473.1,E2 -473.1} C_VEL
LIN {X 0,Y 608.472,Z 574.687,A -85,B 0,C 180,E1 -475.72,E2 -475.72} C_VEL
LIN {X 0,Y 608.475,Z 574.69,A -85,B 0,C 180,E1 -478.62,E2 -478.62} C_VEL
LIN {X 0,Y 608.444,Z 574.688,A -85,B 0,C 180,E1 -481.317,E2 -481.317} C_VEL
LIN {X 0,Y 608.477,Z 574.685,A -85,B 0,C 180,E1 -483.735,E2 -483.735} C_VEL
LIN {X 0,Y 608.476,Z 574.688,A -85,B 0,C 180,E1 -486.089,E2 -486.089} C_VEL
LIN {X 0,Y 608.464,Z 574.696,A -85,B 0,C 180,E1 -488.587,E2 -488.587} C_VEL
LIN {X 0,Y 608.455,Z 574.687,A -85,B 0,C 180,E1 -491.341,E2 -491.341} C_VEL
LIN {X 0,Y 608.451,Z 574.692,A -85,B 0,C 180,E1 -494.263,E2 -494.263} C_VEL
LIN {X 0,Y 608.451,Z 574.692,A -85,B 0,C 180,E1 -497.04,E2 -497.04} C_VEL
LIN {X 0,Y 608.451,Z 574.687,A -85,B 0,C 180,E1 -499.696,E2 -499.696} C_VEL
LIN {X 0,Y 608.47,Z 574.687,A -85,B 0,C 180,E1 -502.253,E2 -502.253} C_VEL
LIN {X 0,Y 608.469,Z 574.691,A -85,B 0,C 180,E1 -505.09,E2 -505.09} C_VEL
LIN {X 0,Y 608.461,Z 574.685,A -85,B 0,C 180,E1 -507.905,E2 -507.905} C_VEL
LIN {X 0,Y 608.47,Z 574.685,A -85,B 0,C 180,E1 -510.22,E2 -510.22} C_VEL
LIN {X 0,Y 608.482,Z 574.691,A -85,B 0,C 180,E1 -512.789,E2 -512.789} C_VEL
LIN {X 0,Y 608.451,Z 574.691,A -85,B 0,C 180,E1 -515.429,E2 -515.429} C_VEL
LIN {X 0,Y 608.462,Z 574.686,A -85,B 0,C 180,E1 -518.308,E2 -518.308} C_VEL
LIN {X 0,Y 608.448,Z 574.699,A -85,B 0,C 180,E1 -521.13,E2 -521.13} C_VEL
LIN {X 0,Y 608.456,Z 574.687,A -85,B 0,C 180,E1 -523.906,E2 -523.906} C_VEL
LIN {X 0,Y 608.459,Z 574.688,A -85,B 0,C 180,E1 -526.643,E2 -526.643} C_VEL
LIN {X 0,Y 608.464,Z 574.695,A -85,B 0,C 180,E1 -529.35,E2 -529.35} C_VEL
LIN {X 0,Y 608.474,Z 574.685,A -85,B 0,C 180,E1 -532.033,E2 -532.033} C_VEL
LIN {X 0,Y 608.457,Z 574.687,A -85,B 0,C 180,E1 -534.698,E2 -534.698} C_VEL
LIN {X 0,Y 608.482,Z 574.693,A -85,B 0,C 180,E1 -537.352,E2 -537.352} C_VEL
LIN {X 0,Y 608.466,Z 574.687,A -85,B 0,C 180,E1 -540,E2 -540} C_VEL
LIN {X 0,Y 608.483,Z 574.683,A -85,B 0,C 180,E1 -542.648,E2 -542.648} C_VEL
LIN {X 0,Y 608.458,Z 574.693,A -85,B 0,C 180,E1 -545.302,E2 -545.302} C_VEL
LIN {X 0,Y 608.474,Z 574.689,A -85,B 0,C 180,E1 -547.967,E2 -547.967} C_VEL
LIN {X 0,Y 608.452,Z 574.691,A -85,B 0,C 180,E1 -549.47,E2 -549.47} C_VEL
LIN {X 0,Y 607.777,Z 574.776,A -85,B 0,C 180,E1 -550.023,E2 -550.023} C_VEL
LIN {X 0,Y 604.924,Z 575.13,A -85,B 0,C 180,E1 -550.92,E2 -550.92} C_VEL
LIN {X 0,Y 602.52,Z 575.437,A -85,B 0,C 180,E1 -551.642,E2 -551.642} C_VEL
LIN {X 0,Y 601.489,Z 575.557,A -85,B 0,C 180,E1 -552.198,E2 -552.198} C_VEL
LIN {X 0,Y 601.406,Z 575.565,A -85,B 0,C 180,E1 -552.387,E2 -552.387} C_VEL
LIN {X 0,Y 601.421,Z 575.563,A -85,B 0,C 180,E1 -554.897,E2 -554.897} C_VEL
LIN {X 0,Y 601.424,Z 575.563,A -85,B 0,C 180,E1 -556.986,E2 -556.986} C_VEL
LIN {X 0,Y 601.4,Z 575.577,A -85,B 0,C 180,E1 -559.809,E2 -559.809} C_VEL
LIN {X 0,Y 601.403,Z 575.565,A -85,B 0,C 180,E1 -562.606,E2 -562.606} C_VEL
LIN {X 0,Y 601.398,Z 575.565,A -85,B 0,C 180,E1 -564.878,E2 -564.878} C_VEL
LIN {X 0,Y 601.414,Z 575.573,A -85,B 0,C 180,E1 -567.867,E2 -567.867} C_VEL
LIN {X 0,Y 601.438,Z 575.569,A -85,B 0,C 180,E1 -570.163,E2 -570.163} C_VEL
LIN {X 0,Y 601.413,Z 575.565,A -85,B 0,C 180,E1 -572.716,E2 -572.716} C_VEL
LIN {X 0,Y 601.401,Z 575.565,A -85,B 0,C 180,E1 -575.115,E2 -575.115} C_VEL
LIN {X 0,Y 601.429,Z 575.562,A -85,B 0,C 180,E1 -577.419,E2 -577.419} C_VEL
LIN {X 0,Y 601.408,Z 575.572,A -85,B 0,C 180,E1 -579.995,E2 -579.995} C_VEL
LIN {X 0,Y 601.43,Z 575.565,A -85,B 0,C 180,E1 -582.668,E2 -582.668} C_VEL
LIN {X 0,Y 601.417,Z 575.564,A -85,B 0,C 180,E1 -585.483,E2 -585.483} C_VEL
LIN {X 0,Y 601.417,Z 575.573,A -85,B 0,C 180,E1 -588.407,E2 -588.407} C_VEL
LIN {X 0,Y 601.429,Z 575.564,A -85,B 0,C 180,E1 -590.876,E2 -590.876} C_VEL
LIN {X 0,Y 601.437,Z 575.562,A -85,B 0,C 180,E1 -593.734,E2 -593.734} C_VEL
LIN {X 0,Y 601.427,Z 575.569,A -85,B 0,C 180,E1 -596.687,E2 -596.687} C_VEL
LIN {X 0,Y 601.424,Z 575.565,A -85,B 0,C 180,E1 -599.059,E2 -599.059} C_VEL
LIN {X 0,Y 601.432,Z 575.562,A -85,B 0,C 180,E1 -601.374,E2 -601.374} C_VEL
LIN {X 0,Y 601.401,Z 575.565,A -85,B 0,C 180,E1 -603.637,E2 -603.637} C_VEL
LIN {X 0,Y 601.415,Z 575.573,A -85,B 0,C 180,E1 -606.59,E2 -606.59} C_VEL
LIN {X 0,Y 601.428,Z 575.562,A -85,B 0,C 180,E1 -609.479,E2 -609.479} C_VEL
LIN {X 0,Y 601.399,Z 575.569,A -85,B 0,C 180,E1 -612.312,E2 -612.312} C_VEL
LIN {X 0,Y 601.414,Z 575.568,A -85,B 0,C 180,E1 -614.409,E2 -614.409} C_VEL
LIN {X 0,Y 601.42,Z 575.568,A -85,B 0,C 180,E1 -617.172,E2 -617.172} C_VEL
LIN {X 0,Y 601.428,Z 575.562,A -85,B 0,C 180,E1 -619.905,E2 -619.905} C_VEL
LIN {X 0,Y 601.441,Z 575.565,A -85,B 0,C 180,E1 -622.615,E2 -622.615} C_VEL
LIN {X 0,Y 601.418,Z 575.568,A -85,B 0,C 180,E1 -625.308,E2 -625.308} C_VEL
LIN {X 0,Y 601.432,Z 575.561,A -85,B 0,C 180,E1 -627.991,E2 -627.991} C_VEL
LIN {X 0,Y 601.441,Z 575.564,A -85,B 0,C 180,E1 -630.67,E2 -630.67} C_VEL
LIN {X 0,Y 601.434,Z 575.568,A -85,B 0,C 180,E1 -633.349,E2 -633.349} C_VEL
LIN {X 0,Y 601.429,Z 575.562,A -85,B 0,C 180,E1 -636.037,E2 -636.037} C_VEL
LIN {X 0,Y 601.413,Z 575.566,A -85,B 0,C 180,E1 -638.738,E2 -638.738} C_VEL
LIN {X 0,Y 601.436,Z 575.569,A -85,B 0,C 180,E1 -641.458,E2 -641.458} C_VEL
LIN {X 0,Y 601.416,Z 575.563,A -85,B 0,C 180,E1 -644.205,E2 -644.205} C_VEL
LIN {X 0,Y 601.431,Z 575.565,A -85,B 0,C 180,E1 -646.985,E2 -646.985} C_VEL
LIN {X 0,Y 601.406,Z 575.569,A -85,B 0,C 180,E1 -649.809,E2 -649.809} C_VEL
LIN {X 0,Y 601.408,Z 575.565,A -85,B 0,C 180,E1 -652.683,E2 -652.683} C_VEL
LIN {X 0,Y 601.401,Z 575.567,A -85,B 0,C 180,E1 -654.878,E2 -654.878} C_VEL
LIN {X 0,Y 601.446,Z 575.702,A -85,B 0,C 180,E1 -656.923,E2 -656.923} C_VEL
LIN {X 0,Y 601.444,Z 590.572,A -85,B 0,C 180,E1 -659.581,E2 -659.581} C_VEL
LIN {X 0,Y 601.404,Z 603.561,A -85,B 0,C 180,E1 -661.874,E2 -661.874} C_VEL
LIN {X 0,Y 601.667,Z 607.599,A -85,B 0,C 180,E1 -661.944,E2 -661.944} C_VEL
LIN {X 0,Y 601.621,Z 709.716,A -85,B 0,C 180,E1 -663.18,E2 -663.18} C_VEL
LIN {X 0,Y 601.57,Z 723.089,A -85,B 0,C 180,E1 -663.479,E2 -663.479} C_VEL
LIN {X 0,Y 601.556,Z 735.146,A -85,B 0,C 180,E1 -663.88,E2 -663.88} C_VEL
LIN {X 0,Y 601.506,Z 747.156,A -85,B 0,C 180,E1 -664.416,E2 -664.416} C_VEL
LIN {X 0,Y 601.47,Z 758.274,A -85,B 0,C 180,E1 -665.059,E2 -665.059} C_VEL
LIN {X 0,Y 601.457,Z 769.036,A -85,B 0,C 180,E1 -665.84,E2 -665.84} C_VEL
LIN {X 0,Y 601.424,Z 778.516,A -85,B 0,C 180,E1 -666.685,E2 -666.685} C_VEL
LIN {X 0,Y 601.375,Z 787.126,A -85,B 0,C 180,E1 -667.633,E2 -667.633} C_VEL
LIN {X 0,Y 601.38,Z 794.227,A -85,B 0,C 180,E1 -668.594,E2 -668.594} C_VEL
LIN {X 0,Y 601.362,Z 800.994,A -85,B 0,C 180,E1 -669.739,E2 -669.739} C_VEL
LIN {X 0,Y 601.336,Z 806.146,A -85,B 0,C 180,E1 -670.88,E2 -670.88} C_VEL
LIN {X 0,Y 601.358,Z 810.307,A -85,B 0,C 180,E1 -672.175,E2 -672.175} C_VEL
LIN {X 0,Y 601.339,Z 811.486,A -85,B 0,C 180,E1 -672.675,E2 -672.675} C_VEL
LIN {X 0,Y 601.337,Z 813.053,A -85,B 0,C 180,E1 -673.593,E2 -673.593} C_VEL
LIN {X 0,Y 601.325,Z 813.881,A -85,B 0,C 180,E1 -674.526,E2 -674.526} C_VEL
LIN {X 0,Y 601.325,Z 813.907,A -85,B 0,C 180,E1 -675.473,E2 -675.473} C_VEL
LIN {X 0,Y 601.338,Z 813.125,A -85,B 0,C 180,E1 -676.435,E2 -676.435} C_VEL
LIN {X 0,Y 601.338,Z 811.484,A -85,B 0,C 180,E1 -677.415,E2 -677.415} C_VEL
LIN {X 0,Y 601.342,Z 808.895,A -85,B 0,C 180,E1 -678.414,E2 -678.414} C_VEL
LIN {X 0,Y 601.33,Z 805.233,A -85,B 0,C 180,E1 -679.435,E2 -679.435} C_VEL
LIN {X 0,Y 601.353,Z 800.342,A -85,B 0,C 180,E1 -680.473,E2 -680.473} C_VEL
LIN {X 0,Y 601.37,Z 793.972,A -85,B 0,C 180,E1 -681.535,E2 -681.535} C_VEL
LIN {X 0,Y 601.404,Z 786.13,A -85,B 0,C 180,E1 -682.579,E2 -682.579} C_VEL
LIN {X 0,Y 601.414,Z 778.383,A -85,B 0,C 180,E1 -683.418,E2 -683.418} C_VEL
LIN {X 0,Y 601.445,Z 767.972,A -85,B 0,C 180,E1 -684.336,E2 -684.336} C_VEL
LIN {X 0,Y 601.485,Z 757.631,A -85,B 0,C 180,E1 -685.073,E2 -685.073} C_VEL
LIN {X 0,Y 601.529,Z 745.862,A -85,B 0,C 180,E1 -685.737,E2 -685.737} C_VEL
LIN {X 0,Y 601.563,Z 732.941,A -85,B 0,C 180,E1 -686.294,E2 -686.294} C_VEL
LIN {X 0,Y 601.589,Z 719.888,A -85,B 0,C 180,E1 -686.697,E2 -686.697} C_VEL
LIN {X 0,Y 601.616,Z 706.449,A -85,B 0,C 180,E1 -686.958,E2 -686.958} C_VEL
LIN {X 0,Y 601.54,Z 604.706,A -85,B 0,C 180,E1 -688.183,E2 -688.183} C_VEL
LIN {X 0,Y 601.395,Z 603.519,A -85,B 0,C 180,E1 -688.224,E2 -688.224} C_VEL
LIN {X 0,Y 601.476,Z 588.125,A -85,B 0,C 180,E1 -690.943,E2 -690.943} C_VEL
LIN {X 0,Y 601.417,Z 575.566,A -85,B 0,C 180,E1 -693.216,E2 -693.216} C_VEL
LIN {X 0,Y 601.453,Z 575.56,A -85,B 0,C 180,E1 -695.86,E2 -695.86} C_VEL
LIN {X 0,Y 601.407,Z 575.573,A -85,B 0,C 180,E1 -698.761,E2 -698.761} C_VEL
LIN {X 0,Y 601.418,Z 575.563,A -85,B 0,C 180,E1 -701.609,E2 -701.609} C_VEL
LIN {X 0,Y 601.414,Z 575.57,A -85,B 0,C 180,E1 -704.409,E2 -704.409} C_VEL
LIN {X 0,Y 601.423,Z 575.566,A -85,B 0,C 180,E1 -707.172,E2 -707.172} C_VEL
LIN {X 0,Y 601.432,Z 575.562,A -85,B 0,C 180,E1 -709.905,E2 -709.905} C_VEL
LIN {X 0,Y 601.448,Z 575.568,A -85,B 0,C 180,E1 -712.615,E2 -712.615} C_VEL
LIN {X 0,Y 601.433,Z 575.564,A -85,B 0,C 180,E1 -715.308,E2 -715.308} C_VEL
LIN {X 0,Y 601.417,Z 575.563,A -85,B 0,C 180,E1 -717.991,E2 -717.991} C_VEL
LIN {X 0,Y 601.45,Z 575.566,A -85,B 0,C 180,E1 -720.67,E2 -720.67} C_VEL
LIN {X 0,Y 601.43,Z 575.565,A -85,B 0,C 180,E1 -723.35,E2 -723.35} C_VEL
LIN {X 0,Y 601.426,Z 575.562,A -85,B 0,C 180,E1 -726.037,E2 -726.037} C_VEL
LIN {X 0,Y 601.438,Z 575.567,A -85,B 0,C 180,E1 -728.738,E2 -728.738} C_VEL
LIN {X 0,Y 601.431,Z 575.565,A -85,B 0,C 180,E1 -731.459,E2 -731.459} C_VEL
LIN {X 0,Y 601.41,Z 575.564,A -85,B 0,C 180,E1 -734.206,E2 -734.206} C_VEL
LIN {X 0,Y 601.428,Z 575.571,A -85,B 0,C 180,E1 -736.986,E2 -736.986} C_VEL
LIN {X 0,Y 601.405,Z 575.566,A -85,B 0,C 180,E1 -739.81,E2 -739.81} C_VEL
LIN {X 0,Y 601.404,Z 575.568,A -85,B 0,C 180,E1 -742.684,E2 -742.684} C_VEL
LIN {X 0,Y 601.4,Z 575.571,A -85,B 0,C 180,E1 -744.879,E2 -744.879} C_VEL
LIN {X 0,Y 601.417,Z 575.565,A -85,B 0,C 180,E1 -747.868,E2 -747.868} C_VEL
LIN {X 0,Y 601.441,Z 575.56,A -85,B 0,C 180,E1 -750.164,E2 -750.164} C_VEL
LIN {X 0,Y 601.417,Z 575.565,A -85,B 0,C 180,E1 -752.717,E2 -752.717} C_VEL
LIN {X 0,Y 601.405,Z 575.572,A -85,B 0,C 180,E1 -755.115,E2 -755.115} C_VEL
LIN {X 0,Y 601.433,Z 575.572,A -85,B 0,C 180,E1 -757.42,E2 -757.42} C_VEL
LIN {X 0,Y 601.41,Z 575.566,A -85,B 0,C 180,E1 -759.995,E2 -759.995} C_VEL
LIN {X 0,Y 601.41,Z 575.565,A -85,B 0,C 180,E1 -762.671,E2 -762.671} C_VEL
LIN {X 0,Y 601.422,Z 575.574,A -85,B 0,C 180,E1 -765.483,E2 -765.483} C_VEL
LIN {X 0,Y 601.42,Z 575.563,A -85,B 0,C 180,E1 -768.408,E2 -768.408} C_VEL
LIN {X 0,Y 601.431,Z 575.563,A -85,B 0,C 180,E1 -770.876,E2 -770.876} C_VEL
LIN {X 0,Y 601.442,Z 575.569,A -85,B 0,C 180,E1 -773.735,E2 -773.735} C_VEL
LIN {X 0,Y 601.429,Z 575.562,A -85,B 0,C 180,E1 -776.688,E2 -776.688} C_VEL
LIN {X 0,Y 601.411,Z 575.566,A -85,B 0,C 180,E1 -779.058,E2 -779.058} C_VEL
LIN {X 0,Y 601.433,Z 575.567,A -85,B 0,C 180,E1 -781.374,E2 -781.374} C_VEL
LIN {X 0,Y 601.411,Z 575.569,A -85,B 0,C 180,E1 -784.134,E2 -784.134} C_VEL
LIN {X 0,Y 601.426,Z 575.655,A -85,B 0,C 180,E1 -786.75,E2 -786.75} C_VEL
LIN {X 0,Y 601.713,Z 580.671,A -85,B 0,C 180,E1 -787.447,E2 -787.447} C_VEL
LIN {X 0,Y 601.592,Z 599.754,A -85,B 0,C 180,E1 -790.02,E2 -790.02} C_VEL
LIN {X 0,Y 601.558,Z 619.698,A -85,B 0,C 180,E1 -792.668,E2 -792.668} C_VEL
LIN {X 0,Y 601.475,Z 642.3,A -85,B 0,C 180,E1 -795.624,E2 -795.624} C_VEL
LIN {X 0,Y 601.456,Z 651.524,A -85,B 0,C 180,E1 -796.819,E2 -796.819} C_VEL
LIN {X 0,Y 601.663,Z 664.691,A -85,B 0,C 180,E1 -796.984,E2 -796.984} C_VEL
LIN {X 0,Y 601.6,Z 759.963,A -85,B 0,C 180,E1 -798.14,E2 -798.14} C_VEL
LIN {X 0,Y 601.58,Z 773.227,A -85,B 0,C 180,E1 -798.438,E2 -798.438} C_VEL
LIN {X 0,Y 601.575,Z 785.666,A -85,B 0,C 180,E1 -798.855,E2 -798.855} C_VEL
LIN {X 0,Y 601.524,Z 797.639,A -85,B 0,C 180,E1 -799.396,E2 -799.396} C_VEL
LIN {X 0,Y 601.477,Z 809.202,A -85,B 0,C 180,E1 -800.076,E2 -800.076} C_VEL
LIN {X 0,Y 601.444,Z 819.597,A -85,B 0,C 180,E1 -800.839,E2 -800.839} C_VEL
LIN {X 0,Y 601.429,Z 828.114,A -85,B 0,C 180,E1 -801.601,E2 -801.601} C_VEL
LIN {X 0,Y 601.418,Z 835.962,A -85,B 0,C 180,E1 -802.446,E2 -802.446} C_VEL
LIN {X 0,Y 601.37,Z 843.226,A -85,B 0,C 180,E1 -803.398,E2 -803.398} C_VEL
LIN {X 0,Y 601.372,Z 848.867,A -85,B 0,C 180,E1 -804.299,E2 -804.299} C_VEL
LIN {X 0,Y 601.336,Z 853.951,A -85,B 0,C 180,E1 -805.307,E2 -805.307} C_VEL
LIN {X 0,Y 601.368,Z 857.896,A -85,B 0,C 180,E1 -806.315,E2 -806.315} C_VEL
LIN {X 0,Y 601.325,Z 860.809,A -85,B 0,C 180,E1 -807.321,E2 -807.321} C_VEL
LIN {X 0,Y 601.34,Z 862.202,A -85,B 0,C 180,E1 -807.991,E2 -807.991} C_VEL
LIN {X 0,Y 601.339,Z 863.784,A -85,B 0,C 180,E1 -809.33,E2 -809.33} C_VEL
LIN {X 0,Y 601.335,Z 864,A -85,B 0,C 180,E1 -810,E2 -810} C_VEL
LIN {X 0,Y 601.348,Z 863.184,A -85,B 0,C 180,E1 -811.339,E2 -811.339} C_VEL
LIN {X 0,Y 601.34,Z 862.202,A -85,B 0,C 180,E1 -812.009,E2 -812.009} C_VEL
LIN {X 0,Y 601.325,Z 860.809,A -85,B 0,C 180,E1 -812.679,E2 -812.679} C_VEL
LIN {X 0,Y 601.368,Z 857.896,A -85,B 0,C 180,E1 -813.685,E2 -813.685} C_VEL
LIN {X 0,Y 601.336,Z 853.95,A -85,B 0,C 180,E1 -814.693,E2 -814.693} C_VEL
LIN {X 0,Y 601.372,Z 847.878,A -85,B 0,C 180,E1 -815.869,E2 -815.869} C_VEL
LIN {X 0,Y 601.382,Z 841.237,A -85,B 0,C 180,E1 -816.88,E2 -816.88} C_VEL
LIN {X 0,Y 601.4,Z 832.991,A -85,B 0,C 180,E1 -817.892,E2 -817.892} C_VEL
LIN {X 0,Y 601.436,Z 824.539,A -85,B 0,C 180,E1 -818.737,E2 -818.737} C_VEL
LIN {X 0,Y 601.44,Z 814.095,A -85,B 0,C 180,E1 -819.585,E2 -819.585} C_VEL
LIN {X 0,Y 601.489,Z 803.761,A -85,B 0,C 180,E1 -820.264,E2 -820.264} C_VEL
LIN {X 0,Y 601.536,Z 792.906,A -85,B 0,C 180,E1 -820.836,E2 -820.836} C_VEL
LIN {X 0,Y 601.566,Z 780.384,A -85,B 0,C 180,E1 -821.34,E2 -821.34} C_VEL
LIN {X 0,Y 601.595,Z 767.365,A -85,B 0,C 180,E1 -821.711,E2 -821.711} C_VEL
LIN {X 0,Y 601.608,Z 754.107,A -85,B 0,C 180,E1 -821.946,E2 -821.946} C_VEL
LIN {X 0,Y 601.535,Z 652.17,A -85,B 0,C 180,E1 -823.169,E2 -823.169} C_VEL
LIN {X 0,Y 601.473,Z 651.275,A -85,B 0,C 180,E1 -823.213,E2 -823.213} C_VEL
LIN {X 0,Y 601.515,Z 629.005,A -85,B 0,C 180,E1 -826.11,E2 -826.11} C_VEL
LIN {X 0,Y 601.558,Z 608.178,A -85,B 0,C 180,E1 -828.857,E2 -828.857} C_VEL
LIN {X 0,Y 601.67,Z 587.788,A -85,B 0,C 180,E1 -831.588,E2 -831.588} C_VEL
LIN {X 0,Y 601.687,Z 577.151,A -85,B 0,C 180,E1 -833.035,E2 -833.035} C_VEL
LIN {X 0,Y 601.414,Z 575.568,A -85,B 0,C 180,E1 -833.273,E2 -833.273} C_VEL
LIN {X 0,Y 601.413,Z 575.568,A -85,B 0,C 180,E1 -835.867,E2 -835.867} C_VEL
LIN {X 0,Y 601.434,Z 575.567,A -85,B 0,C 180,E1 -838.626,E2 -838.626} C_VEL
LIN {X 0,Y 601.419,Z 575.563,A -85,B 0,C 180,E1 -841.454,E2 -841.454} C_VEL
LIN {X 0,Y 601.431,Z 575.567,A -85,B 0,C 180,E1 -844.117,E2 -844.117} C_VEL
LIN {X 0,Y 601.409,Z 575.574,A -85,B 0,C 180,E1 -846.581,E2 -846.581} C_VEL
LIN {X 0,Y 601.438,Z 575.56,A -85,B 0,C 180,E1 -849.535,E2 -849.535} C_VEL
LIN {X 0,Y 601.409,Z 575.576,A -85,B 0,C 180,E1 -852.59,E2 -852.59} C_VEL
LIN {X 0,Y 601.421,Z 575.563,A -85,B 0,C 180,E1 -855.481,E2 -855.481} C_VEL
LIN {X 0,Y 601.425,Z 575.568,A -85,B 0,C 180,E1 -858.405,E2 -858.405} C_VEL
LIN {X 0,Y 601.434,Z 575.57,A -85,B 0,C 180,E1 -860.875,E2 -860.875} C_VEL
LIN {X 0,Y 601.438,Z 575.56,A -85,B 0,C 180,E1 -863.733,E2 -863.733} C_VEL
LIN {X 0,Y 601.424,Z 575.57,A -85,B 0,C 180,E1 -866.686,E2 -866.686} C_VEL
LIN {X 0,Y 601.427,Z 575.57,A -85,B 0,C 180,E1 -869.058,E2 -869.058} C_VEL
LIN {X 0,Y 601.425,Z 575.566,A -85,B 0,C 180,E1 -871.372,E2 -871.372} C_VEL
LIN {X 0,Y 601.4,Z 575.566,A -85,B 0,C 180,E1 -873.636,E2 -873.636} C_VEL
LIN {X 0,Y 601.418,Z 575.567,A -85,B 0,C 180,E1 -876.589,E2 -876.589} C_VEL
LIN {X 0,Y 601.426,Z 575.566,A -85,B 0,C 180,E1 -879.478,E2 -879.478} C_VEL
LIN {X 0,Y 601.394,Z 575.566,A -85,B 0,C 180,E1 -882.311,E2 -882.311} C_VEL
LIN {X 0,Y 601.407,Z 575.565,A -85,B 0,C 180,E1 -884.408,E2 -884.408} C_VEL
LIN {X 0,Y 601.418,Z 575.573,A -85,B 0,C 180,E1 -887.171,E2 -887.171} C_VEL
LIN {X 0,Y 601.432,Z 575.563,A -85,B 0,C 180,E1 -889.905,E2 -889.905} C_VEL
LIN {X 0,Y 601.444,Z 575.561,A -85,B 0,C 180,E1 -892.615,E2 -892.615} C_VEL
LIN {X 0,Y 601.431,Z 575.572,A -85,B 0,C 180,E1 -895.308,E2 -895.308} C_VEL
LIN {X 0,Y 601.416,Z 575.565,A -85,B 0,C 180,E1 -897.991,E2 -897.991} C_VEL
LIN {X 0,Y 601.449,Z 575.56,A -85,B 0,C 180,E1 -900.669,E2 -900.669} C_VEL
LIN {X 0,Y 601.427,Z 575.57,A -85,B 0,C 180,E1 -903.349,E2 -903.349} C_VEL
LIN {X 0,Y 601.406,Z 575.568,A -85,B 0,C 180,E1 -906.037,E2 -906.037} C_VEL
LIN {X 0,Y 601.435,Z 575.561,A -85,B 0,C 180,E1 -908.737,E2 -908.737} C_VEL
LIN {X 0,Y 601.426,Z 575.569,A -85,B 0,C 180,E1 -911.458,E2 -911.458} C_VEL
LIN {X 0,Y 601.406,Z 575.565,A -85,B 0,C 180,E1 -912.387,E2 -912.387} C_VEL
LIN {X 0,Y 600.74,Z 575.649,A -85,B 0,C 180,E1 -912.946,E2 -912.946} C_VEL
LIN {X 0,Y 597.887,Z 576.011,A -85,B 0,C 180,E1 -913.854,E2 -913.854} C_VEL
LIN {X 0,Y 595.475,Z 576.307,A -85,B 0,C 180,E1 -914.584,E2 -914.584} C_VEL
LIN {X 0,Y 594.439,Z 576.435,A -85,B 0,C 180,E1 -915.148,E2 -915.148} C_VEL
LIN {X 0,Y 594.354,Z 576.447,A -85,B 0,C 180,E1 -915.338,E2 -915.338} C_VEL
LIN {X 0,Y 594.374,Z 576.449,A -85,B 0,C 180,E1 -917.904,E2 -917.904} C_VEL
LIN {X 0,Y 594.374,Z 576.44,A -85,B 0,C 180,E1 -920.919,E2 -920.919} C_VEL
LIN {X 0,Y 594.386,Z 576.447,A -85,B 0,C 180,E1 -923.704,E2 -923.704} C_VEL
LIN {X 0,Y 594.379,Z 576.44,A -85,B 0,C 180,E1 -926.699,E2 -926.699} C_VEL
LIN {X 0,Y 594.372,Z 576.441,A -85,B 0,C 180,E1 -928.998,E2 -928.998} C_VEL
LIN {X 0,Y 594.383,Z 576.444,A -85,B 0,C 180,E1 -931.646,E2 -931.646} C_VEL
LIN {X 0,Y 594.385,Z 576.442,A -85,B 0,C 180,E1 -934.579,E2 -934.579} C_VEL
LIN {X 0,Y 594.38,Z 576.44,A -85,B 0,C 180,E1 -937.087,E2 -937.087} C_VEL
LIN {X 0,Y 594.371,Z 576.445,A -85,B 0,C 180,E1 -939.775,E2 -939.775} C_VEL
LIN {X 0,Y 594.38,Z 576.448,A -85,B 0,C 180,E1 -942.374,E2 -942.374} C_VEL
LIN {X 0,Y 594.354,Z 576.443,A -85,B 0,C 180,E1 -945.192,E2 -945.192} C_VEL
LIN {X 0,Y 594.361,Z 576.443,A -85,B 0,C 180,E1 -947.625,E2 -947.625} C_VEL
LIN {X 0,Y 594.386,Z 576.45,A -85,B 0,C 180,E1 -950.322,E2 -950.322} C_VEL
LIN {X 0,Y 594.379,Z 576.443,A -85,B 0,C 180,E1 -952.914,E2 -952.914} C_VEL
LIN {X 0,Y 594.381,Z 576.441,A -85,B 0,C 180,E1 -955.861,E2 -955.861} C_VEL
LIN {X 0,Y 594.385,Z 576.448,A -85,B 0,C 180,E1 -958.652,E2 -958.652} C_VEL
LIN {X 0,Y 594.38,Z 576.443,A -85,B 0,C 180,E1 -961.042,E2 -961.042} C_VEL
LIN {X 0,Y 594.383,Z 576.441,A -85,B 0,C 180,E1 -963.977,E2 -963.977} C_VEL
LIN {X 0,Y 594.385,Z 576.444,A -85,B 0,C 180,E1 -966.296,E2 -966.296} C_VEL
LIN {X 0,Y 594.401,Z 576.44,A -85,B 0,C 180,E1 -969.225,E2 -969.225} C_VEL
LIN {X 0,Y 594.377,Z 576.441,A -85,B 0,C 180,E1 -972.096,E2 -972.096} C_VEL
LIN {X 0,Y 594.367,Z 576.443,A -85,B 0,C 180,E1 -974.219,E2 -974.219} C_VEL
LIN {X 0,Y 594.368,Z 576.449,A -85,B 0,C 180,E1 -977.017,E2 -977.017} C_VEL
LIN {X 0,Y 594.388,Z 576.439,A -85,B 0,C 180,E1 -979.784,E2 -979.784} C_VEL
LIN {X 0,Y 594.393,Z 576.442,A -85,B 0,C 180,E1 -982.527,E2 -982.527} C_VEL
LIN {X 0,Y 594.388,Z 576.445,A -85,B 0,C 180,E1 -985.252,E2 -985.252} C_VEL
LIN {X 0,Y 594.401,Z 576.437,A -85,B 0,C 180,E1 -987.967,E2 -987.967} C_VEL
LIN {X 0,Y 594.413,Z 576.439,A -85,B 0,C 180,E1 -990.677,E2 -990.677} C_VEL
LIN {X 0,Y 594.385,Z 576.446,A -85,B 0,C 180,E1 -993.389,E2 -993.389} C_VEL
LIN {X 0,Y 594.379,Z 576.44,A -85,B 0,C 180,E1 -996.109,E2 -996.109} C_VEL
LIN {X 0,Y 594.38,Z 576.444,A -85,B 0,C 180,E1 -998.842,E2 -998.842} C_VEL
LIN {X 0,Y 594.394,Z 576.444,A -85,B 0,C 180,E1 -1001.595,E2 -1001.595} C_VEL
LIN {X 0,Y 594.386,Z 576.439,A -85,B 0,C 180,E1 -1004.377,E2 -1004.377} C_VEL
LIN {X 0,Y 594.389,Z 576.446,A -85,B 0,C 180,E1 -1007.193,E2 -1007.193} C_VEL
LIN {X 0,Y 594.374,Z 576.443,A -85,B 0,C 180,E1 -1010.053,E2 -1010.053} C_VEL
LIN {X 0,Y 594.36,Z 576.445,A -85,B 0,C 180,E1 -1012.967,E2 -1012.967} C_VEL
LIN {X 0,Y 594.379,Z 576.446,A -85,B 0,C 180,E1 -1015.192,E2 -1015.192} C_VEL
LIN {X 0,Y 594.39,Z 576.474,A -85,B 0,C 180,E1 -1016.841,E2 -1016.841} C_VEL
LIN {X 0,Y 594.43,Z 590.514,A -85,B 0,C 180,E1 -1019.383,E2 -1019.383} C_VEL
LIN {X 0,Y 594.36,Z 603.581,A -85,B 0,C 180,E1 -1021.718,E2 -1021.718} C_VEL
LIN {X 0,Y 594.77,Z 607.96,A -85,B 0,C 180,E1 -1021.794,E2 -1021.794} C_VEL
LIN {X 0,Y 594.671,Z 710.284,A -85,B 0,C 180,E1 -1023.05,E2 -1023.05} C_VEL
LIN {X 0,Y 594.619,Z 723.852,A -85,B 0,C 180,E1 -1023.364,E2 -1023.364} C_VEL
LIN {X 0,Y 594.587,Z 737.006,A -85,B 0,C 180,E1 -1023.82,E2 -1023.82} C_VEL
LIN {X 0,Y 594.507,Z 748.744,A -85,B 0,C 180,E1 -1024.375,E2 -1024.375} C_VEL
LIN {X 0,Y 594.427,Z 760.295,A -85,B 0,C 180,E1 -1025.076,E2 -1025.076} C_VEL
LIN {X 0,Y 594.427,Z 770.142,A -85,B 0,C 180,E1 -1025.819,E2 -1025.819} C_VEL
LIN {X 0,Y 594.375,Z 778.596,A -85,B 0,C 180,E1 -1026.593,E2 -1026.593} C_VEL
LIN {X 0,Y 594.299,Z 787.549,A -85,B 0,C 180,E1 -1027.598,E2 -1027.598} C_VEL
LIN {X 0,Y 594.304,Z 795.4,A -85,B 0,C 180,E1 -1028.695,E2 -1028.695} C_VEL
LIN {X 0,Y 594.281,Z 801.45,A -85,B 0,C 180,E1 -1029.764,E2 -1029.764} C_VEL
LIN {X 0,Y 594.238,Z 806.062,A -85,B 0,C 180,E1 -1030.807,E2 -1030.807} C_VEL
LIN {X 0,Y 594.266,Z 809.51,A -85,B 0,C 180,E1 -1031.836,E2 -1031.836} C_VEL
LIN {X 0,Y 594.244,Z 811.894,A -85,B 0,C 180,E1 -1032.84,E2 -1032.84} C_VEL
LIN {X 0,Y 594.222,Z 813.703,A -85,B 0,C 180,E1 -1034.25,E2 -1034.25} C_VEL
LIN {X 0,Y 594.21,Z 813.969,A -85,B 0,C 180,E1 -1035.205,E2 -1035.205} C_VEL
LIN {X 0,Y 594.229,Z 813.445,A -85,B 0,C 180,E1 -1036.173,E2 -1036.173} C_VEL
LIN {X 0,Y 594.243,Z 812.068,A -85,B 0,C 180,E1 -1037.159,E2 -1037.159} C_VEL
LIN {X 0,Y 594.238,Z 808.677,A -85,B 0,C 180,E1 -1038.525,E2 -1038.525} C_VEL
LIN {X 0,Y 594.25,Z 805.497,A -85,B 0,C 180,E1 -1039.424,E2 -1039.424} C_VEL
LIN {X 0,Y 594.291,Z 800.365,A -85,B 0,C 180,E1 -1040.533,E2 -1040.533} C_VEL
LIN {X 0,Y 594.296,Z 793.535,A -85,B 0,C 180,E1 -1041.679,E2 -1041.679} C_VEL
LIN {X 0,Y 594.352,Z 786.216,A -85,B 0,C 180,E1 -1042.659,E2 -1042.659} C_VEL
LIN {X 0,Y 594.408,Z 777.124,A -85,B 0,C 180,E1 -1043.64,E2 -1043.64} C_VEL
LIN {X 0,Y 594.416,Z 767.413,A -85,B 0,C 180,E1 -1044.492,E2 -1044.492} C_VEL
LIN {X 0,Y 594.465,Z 757.212,A -85,B 0,C 180,E1 -1045.22,E2 -1045.22} C_VEL
LIN {X 0,Y 594.535,Z 746.4,A -85,B 0,C 180,E1 -1045.838,E2 -1045.838} C_VEL
LIN {X 0,Y 594.588,Z 733.522,A -85,B 0,C 180,E1 -1046.406,E2 -1046.406} C_VEL
LIN {X 0,Y 594.633,Z 720.693,A -85,B 0,C 180,E1 -1046.815,E2 -1046.815} C_VEL
LIN {X 0,Y 594.675,Z 707.671,A -85,B 0,C 180,E1 -1047.081,E2 -1047.081} C_VEL
LIN {X 0,Y 594.666,Z 605.52,A -85,B 0,C 180,E1 -1048.328,E2 -1048.328} C_VEL
LIN {X 0,Y 594.357,Z 603.657,A -85,B 0,C 180,E1 -1048.358,E2 -1048.358} C_VEL
LIN {X 0,Y 594.445,Z 587.683,A -85,B 0,C 180,E1 -1051.216,E2 -1051.216} C_VEL
LIN {X 0,Y 594.386,Z 576.443,A -85,B 0,C 180,E1 -1053.277,E2 -1053.277} C_VEL
LIN {X 0,Y 594.387,Z 576.446,A -85,B 0,C 180,E1 -1056.296,E2 -1056.296} C_VEL
LIN {X 0,Y 594.398,Z 576.439,A -85,B 0,C 180,E1 -1059.225,E2 -1059.225} C_VEL
LIN {X 0,Y 594.379,Z 576.443,A -85,B 0,C 180,E1 -1062.096,E2 -1062.096} C_VEL
LIN {X 0,Y 594.365,Z 576.445,A -85,B 0,C 180,E1 -1064.219,E2 -1064.219} C_VEL
LIN {X 0,Y 594.37,Z 576.447,A -85,B 0,C 180,E1 -1067.017,E2 -1067.017} C_VEL
LIN {X 0,Y 594.391,Z 576.439,A -85,B 0,C 180,E1 -1069.784,E2 -1069.784} C_VEL
LIN {X 0,Y 594.411,Z 576.443,A -85,B 0,C 180,E1 -1072.527,E2 -1072.527} C_VEL
LIN {X 0,Y 594.401,Z 576.441,A -85,B 0,C 180,E1 -1075.253,E2 -1075.253} C_VEL
LIN {X 0,Y 594.387,Z 576.439,A -85,B 0,C 180,E1 -1077.968,E2 -1077.968} C_VEL
LIN {X 0,Y 594.42,Z 576.442,A -85,B 0,C 180,E1 -1080.678,E2 -1080.678} C_VEL
LIN {X 0,Y 594.381,Z 576.443,A -85,B 0,C 180,E1 -1083.39,E2 -1083.39} C_VEL
LIN {X 0,Y 594.38,Z 576.44,A -85,B 0,C 180,E1 -1086.109,E2 -1086.109} C_VEL
LIN {X 0,Y 594.398,Z 576.446,A -85,B 0,C 180,E1 -1088.842,E2 -1088.842} C_VEL
LIN {X 0,Y 594.389,Z 576.441,A -85,B 0,C 180,E1 -1091.596,E2 -1091.596} C_VEL
LIN {X 0,Y 594.38,Z 576.441,A -85,B 0,C 180,E1 -1094.378,E2 -1094.378} C_VEL
LIN {X 0,Y 594.386,Z 576.449,A -85,B 0,C 180,E1 -1097.194,E2 -1097.194} C_VEL
LIN {X 0,Y 594.373,Z 576.441,A -85,B 0,C 180,E1 -1100.054,E2 -1100.054} C_VEL
LIN {X 0,Y 594.358,Z 576.45,A -85,B 0,C 180,E1 -1102.968,E2 -1102.968} C_VEL
LIN {X 0,Y 594.374,Z 576.452,A -85,B 0,C 180,E1 -1105.193,E2 -1105.193} C_VEL
LIN {X 0,Y 594.377,Z 576.446,A -85,B 0,C 180,E1 -1107.528,E2 -1107.528} C_VEL
LIN {X 0,Y 594.394,Z 576.438,A -85,B 0,C 180,E1 -1110.332,E2 -1110.332} C_VEL
LIN {X 0,Y 594.373,Z 576.445,A -85,B 0,C 180,E1 -1112.951,E2 -1112.951} C_VEL
LIN {X 0,Y 594.376,Z 576.45,A -85,B 0,C 180,E1 -1115.408,E2 -1115.408} C_VEL
LIN {X 0,Y 594.387,Z 576.441,A -85,B 0,C 180,E1 -1117.941,E2 -1117.941} C_VEL
LIN {X 0,Y 594.377,Z 576.442,A -85,B 0,C 180,E1 -1120.824,E2 -1120.824} C_VEL
LIN {X 0,Y 594.378,Z 576.445,A -85,B 0,C 180,E1 -1123.842,E2 -1123.842} C_VEL
LIN {X 0,Y 594.363,Z 576.443,A -85,B 0,C 180,E1 -1126.702,E2 -1126.702} C_VEL
LIN {X 0,Y 594.368,Z 576.451,A -85,B 0,C 180,E1 -1129.434,E2 -1129.434} C_VEL
LIN {X 0,Y 594.387,Z 576.44,A -85,B 0,C 180,E1 -1132.392,E2 -1132.392} C_VEL
LIN {X 0,Y 594.383,Z 576.44,A -85,B 0,C 180,E1 -1134.673,E2 -1134.673} C_VEL
LIN {X 0,Y 594.38,Z 576.443,A -85,B 0,C 180,E1 -1137.089,E2 -1137.089} C_VEL
LIN {X 0,Y 594.385,Z 576.451,A -85,B 0,C 180,E1 -1139.673,E2 -1139.673} C_VEL
LIN {X 0,Y 594.375,Z 576.441,A -85,B 0,C 180,E1 -1142.54,E2 -1142.54} C_VEL
LIN {X 0,Y 594.374,Z 576.442,A -85,B 0,C 180,E1 -1144.808,E2 -1144.808} C_VEL
LIN {X 0,Y 594.392,Z 576.486,A -85,B 0,C 180,E1 -1146.574,E2 -1146.574} C_VEL
LIN {X 0,Y 594.798,Z 580.644,A -85,B 0,C 180,E1 -1147.166,E2 -1147.166} C_VEL
LIN {X 0,Y 594.694,Z 599.754,A -85,B 0,C 180,E1 -1149.778,E2 -1149.778} C_VEL
LIN {X 0,Y 594.588,Z 621.027,A -85,B 0,C 180,E1 -1152.636,E2 -1152.636} C_VEL
LIN {X 0,Y 594.471,Z 643.63,A -85,B 0,C 180,E1 -1155.625,E2 -1155.625} C_VEL
LIN {X 0,Y 594.466,Z 651.524,A -85,B 0,C 180,E1 -1156.661,E2 -1156.661} C_VEL
LIN {X 0,Y 594.762,Z 657.536,A -85,B 0,C 180,E1 -1156.744,E2 -1156.744} C_VEL
LIN {X 0,Y 594.68,Z 759.963,A -85,B 0,C 180,E1 -1158,E2 -1158} C_VEL
LIN {X 0,Y 594.643,Z 773.228,A -85,B 0,C 180,E1 -1158.301,E2 -1158.301} C_VEL
LIN {X 0,Y 594.59,Z 786.384,A -85,B 0,C 180,E1 -1158.75,E2 -1158.75} C_VEL
LIN {X 0,Y 594.538,Z 797.638,A -85,B 0,C 180,E1 -1159.27,E2 -1159.27} C_VEL
LIN {X 0,Y 594.472,Z 809.203,A -85,B 0,C 180,E1 -1159.958,E2 -1159.958} C_VEL
LIN {X 0,Y 594.413,Z 819.599,A -85,B 0,C 180,E1 -1160.73,E2 -1160.73} C_VEL
LIN {X 0,Y 594.383,Z 828.114,A -85,B 0,C 180,E1 -1161.501,E2 -1161.501} C_VEL
LIN {X 0,Y 594.347,Z 835.962,A -85,B 0,C 180,E1 -1162.356,E2 -1162.356} C_VEL
LIN {X 0,Y 594.282,Z 843.814,A -85,B 0,C 180,E1 -1163.409,E2 -1163.409} C_VEL
LIN {X 0,Y 594.289,Z 850.681,A -85,B 0,C 180,E1 -1164.571,E2 -1164.571} C_VEL
LIN {X 0,Y 594.271,Z 855.372,A -85,B 0,C 180,E1 -1165.591,E2 -1165.591} C_VEL
LIN {X 0,Y 594.268,Z 858.956,A -85,B 0,C 180,E1 -1166.61,E2 -1166.61} C_VEL
LIN {X 0,Y 594.226,Z 860.809,A -85,B 0,C 180,E1 -1167.288,E2 -1167.288} C_VEL
LIN {X 0,Y 594.239,Z 862.202,A -85,B 0,C 180,E1 -1167.967,E2 -1167.967} C_VEL
LIN {X 0,Y 594.239,Z 863.784,A -85,B 0,C 180,E1 -1169.322,E2 -1169.322} C_VEL
LIN {X 0,Y 594.236,Z 864,A -85,B 0,C 180,E1 -1170,E2 -1170} C_VEL
LIN {X 0,Y 594.247,Z 863.185,A -85,B 0,C 180,E1 -1171.355,E2 -1171.355} C_VEL
LIN {X 0,Y 594.239,Z 862.202,A -85,B 0,C 180,E1 -1172.033,E2 -1172.033} C_VEL
LIN {X 0,Y 594.226,Z 860.81,A -85,B 0,C 180,E1 -1172.712,E2 -1172.712} C_VEL
LIN {X 0,Y 594.289,Z 857.896,A -85,B 0,C 180,E1 -1173.729,E2 -1173.729} C_VEL
LIN {X 0,Y 594.241,Z 853.95,A -85,B 0,C 180,E1 -1174.749,E2 -1174.749} C_VEL
LIN {X 0,Y 594.304,Z 847.878,A -85,B 0,C 180,E1 -1175.939,E2 -1175.939} C_VEL
LIN {X 0,Y 594.308,Z 841.237,A -85,B 0,C 180,E1 -1176.962,E2 -1176.962} C_VEL
LIN {X 0,Y 594.359,Z 832.991,A -85,B 0,C 180,E1 -1177.986,E2 -1177.986} C_VEL
LIN {X 0,Y 594.382,Z 824.539,A -85,B 0,C 180,E1 -1178.842,E2 -1178.842} C_VEL
LIN {X 0,Y 594.423,Z 814.096,A -85,B 0,C 180,E1 -1179.699,E2 -1179.699} C_VEL
LIN {X 0,Y 594.489,Z 803.762,A -85,B 0,C 180,E1 -1180.386,E2 -1180.386} C_VEL
LIN {X 0,Y 594.56,Z 792.706,A -85,B 0,C 180,E1 -1180.974,E2 -1180.974} C_VEL
LIN {X 0,Y 594.602,Z 780.712,A -85,B 0,C 180,E1 -1181.464,E2 -1181.464} C_VEL
LIN {X 0,Y 594.64,Z 767.364,A -85,B 0,C 180,E1 -1181.85,E2 -1181.85} C_VEL
LIN {X 0,Y 594.685,Z 754.107,A -85,B 0,C 180,E1 -1182.087,E2 -1182.087} C_VEL
LIN {X 0,Y 594.655,Z 653.065,A -85,B 0,C 180,E1 -1183.313,E2 -1183.313} C_VEL
LIN {X 0,Y 594.453,Z 651.441,A -85,B 0,C 180,E1 -1183.35,E2 -1183.35} C_VEL
LIN {X 0,Y 594.541,Z 629.005,A -85,B 0,C 180,E1 -1186.304,E2 -1186.304} C_VEL
LIN {X 0,Y 594.635,Z 608.076,A -85,B 0,C 180,E1 -1189.099,E2 -1189.099} C_VEL
LIN {X 0,Y 594.769,Z 587.788,A -85,B 0,C 180,E1 -1191.852,E2 -1191.852} C_VEL
LIN {X 0,Y 594.758,Z 578.481,A -85,B 0,C 180,E1 -1193.135,E2 -1193.135} C_VEL
LIN {X 0,Y 594.379,Z 576.446,A -85,B 0,C 180,E1 -1193.45,E2 -1193.45} C_VEL
LIN {X 0,Y 594.388,Z 576.446,A -85,B 0,C 180,E1 -1196.022,E2 -1196.022} C_VEL
LIN {X 0,Y 594.384,Z 576.441,A -85,B 0,C 180,E1 -1198.957,E2 -1198.957} C_VEL
LIN {X 0,Y 594.378,Z 576.441,A -85,B 0,C 180,E1 -1201.642,E2 -1201.642} C_VEL
LIN {X 0,Y 594.393,Z 576.447,A -85,B 0,C 180,E1 -1204.578,E2 -1204.578} C_VEL
LIN {X 0,Y 594.382,Z 576.441,A -85,B 0,C 180,E1 -1207.086,E2 -1207.086} C_VEL
LIN {X 0,Y 594.373,Z 576.441,A -85,B 0,C 180,E1 -1209.774,E2 -1209.774} C_VEL
LIN {X 0,Y 594.366,Z 576.449,A -85,B 0,C 180,E1 -1212.374,E2 -1212.374} C_VEL
LIN {X 0,Y 594.359,Z 576.445,A -85,B 0,C 180,E1 -1215.19,E2 -1215.19} C_VEL
LIN {X 0,Y 594.368,Z 576.441,A -85,B 0,C 180,E1 -1217.624,E2 -1217.624} C_VEL
LIN {X 0,Y 594.389,Z 576.443,A -85,B 0,C 180,E1 -1220.32,E2 -1220.32} C_VEL
LIN {X 0,Y 594.383,Z 576.448,A -85,B 0,C 180,E1 -1222.913,E2 -1222.913} C_VEL
LIN {X 0,Y 594.378,Z 576.44,A -85,B 0,C 180,E1 -1225.86,E2 -1225.86} C_VEL
LIN {X 0,Y 594.385,Z 576.446,A -85,B 0,C 180,E1 -1228.65,E2 -1228.65} C_VEL
LIN {X 0,Y 594.376,Z 576.449,A -85,B 0,C 180,E1 -1231.041,E2 -1231.041} C_VEL
LIN {X 0,Y 594.382,Z 576.439,A -85,B 0,C 180,E1 -1233.975,E2 -1233.975} C_VEL
LIN {X 0,Y 594.387,Z 576.44,A -85,B 0,C 180,E1 -1236.296,E2 -1236.296} C_VEL
LIN {X 0,Y 594.399,Z 576.446,A -85,B 0,C 180,E1 -1239.224,E2 -1239.224} C_VEL
LIN {X 0,Y 594.374,Z 576.44,A -85,B 0,C 180,E1 -1242.095,E2 -1242.095} C_VEL
LIN {X 0,Y 594.361,Z 576.442,A -85,B 0,C 180,E1 -1244.219,E2 -1244.219} C_VEL
LIN {X 0,Y 594.364,Z 576.449,A -85,B 0,C 180,E1 -1247.017,E2 -1247.017} C_VEL
LIN {X 0,Y 594.391,Z 576.441,A -85,B 0,C 180,E1 -1249.784,E2 -1249.784} C_VEL
LIN {X 0,Y 594.393,Z 576.438,A -85,B 0,C 180,E1 -1252.526,E2 -1252.526} C_VEL
LIN {X 0,Y 594.398,Z 576.446,A -85,B 0,C 180,E1 -1255.252,E2 -1255.252} C_VEL
LIN {X 0,Y 594.387,Z 576.441,A -85,B 0,C 180,E1 -1257.967,E2 -1257.967} C_VEL
LIN {X 0,Y 594.419,Z 576.435,A -85,B 0,C 180,E1 -1260.677,E2 -1260.677} C_VEL
LIN {X 0,Y 594.378,Z 576.449,A -85,B 0,C 180,E1 -1263.389,E2 -1263.389} C_VEL
LIN {X 0,Y 594.362,Z 576.444,A -85,B 0,C 180,E1 -1266.109,E2 -1266.109} C_VEL
LIN {X 0,Y 594.394,Z 576.438,A -85,B 0,C 180,E1 -1268.842,E2 -1268.842} C_VEL
LIN {X 0,Y 594.385,Z 576.449,A -85,B 0,C 180,E1 -1271.596,E2 -1271.596} C_VEL
LIN {X 0,Y 594.378,Z 576.441,A -85,B 0,C 180,E1 -1274.377,E2 -1274.377} C_VEL
LIN {X 0,Y 594.354,Z 576.447,A -85,B 0,C 180,E1 -1275.338,E2 -1275.338} C_VEL
LIN {X 0,Y 593.685,Z 576.537,A -85,B 0,C 180,E1 -1275.904,E2 -1275.904} C_VEL
LIN {X 0,Y 590.833,Z 576.893,A -85,B 0,C 180,E1 -1276.822,E2 -1276.822} C_VEL
LIN {X 0,Y 588.427,Z 577.19,A -85,B 0,C 180,E1 -1277.561,E2 -1277.561} C_VEL
LIN {X 0,Y 587.399,Z 577.315,A -85,B 0,C 180,E1 -1278.131,E2 -1278.131} C_VEL
LIN {X 0,Y 587.317,Z 577.322,A -85,B 0,C 180,E1 -1278.324,E2 -1278.324} C_VEL
LIN {X 0,Y 587.346,Z 577.316,A -85,B 0,C 180,E1 -1281.045,E2 -1281.045} C_VEL
LIN {X 0,Y 587.33,Z 577.327,A -85,B 0,C 180,E1 -1284.006,E2 -1284.006} C_VEL
LIN {X 0,Y 587.353,Z 577.32,A -85,B 0,C 180,E1 -1286.277,E2 -1286.277} C_VEL
LIN {X 0,Y 587.341,Z 577.317,A -85,B 0,C 180,E1 -1289.134,E2 -1289.134} C_VEL
LIN {X 0,Y 587.346,Z 577.323,A -85,B 0,C 180,E1 -1291.838,E2 -1291.838} C_VEL
LIN {X 0,Y 587.346,Z 577.322,A -85,B 0,C 180,E1 -1294.349,E2 -1294.349} C_VEL
LIN {X 0,Y 587.344,Z 577.318,A -85,B 0,C 180,E1 -1296.747,E2 -1296.747} C_VEL
LIN {X 0,Y 587.34,Z 577.317,A -85,B 0,C 180,E1 -1299.359,E2 -1299.359} C_VEL
LIN {X 0,Y 587.357,Z 577.324,A -85,B 0,C 180,E1 -1302.112,E2 -1302.112} C_VEL
LIN {X 0,Y 587.306,Z 577.321,A -85,B 0,C 180,E1 -1305.089,E2 -1305.089} C_VEL
LIN {X 0,Y 587.344,Z 577.32,A -85,B 0,C 180,E1 -1307.928,E2 -1307.928} C_VEL
LIN {X 0,Y 587.327,Z 577.319,A -85,B 0,C 180,E1 -1311.058,E2 -1311.058} C_VEL
LIN {X 0,Y 587.347,Z 577.316,A -85,B 0,C 180,E1 -1313.292,E2 -1313.292} C_VEL
LIN {X 0,Y 587.363,Z 577.315,A -85,B 0,C 180,E1 -1315.781,E2 -1315.781} C_VEL
LIN {X 0,Y 587.349,Z 577.322,A -85,B 0,C 180,E1 -1318.232,E2 -1318.232} C_VEL
LIN {X 0,Y 587.346,Z 577.321,A -85,B 0,C 180,E1 -1320.866,E2 -1320.866} C_VEL
LIN {X 0,Y 587.355,Z 577.315,A -85,B 0,C 180,E1 -1323.819,E2 -1323.819} C_VEL
LIN {X 0,Y 587.332,Z 577.319,A -85,B 0,C 180,E1 -1325.994,E2 -1325.994} C_VEL
LIN {X 0,Y 587.321,Z 577.322,A -85,B 0,C 180,E1 -1328.226,E2 -1328.226} C_VEL
LIN {X 0,Y 587.346,Z 577.32,A -85,B 0,C 180,E1 -1331.152,E2 -1331.152} C_VEL
LIN {X 0,Y 587.349,Z 577.318,A -85,B 0,C 180,E1 -1333.312,E2 -1333.312} C_VEL
LIN {X 0,Y 587.359,Z 577.315,A -85,B 0,C 180,E1 -1336.155,E2 -1336.155} C_VEL
LIN {X 0,Y 587.339,Z 577.327,A -85,B 0,C 180,E1 -1338.963,E2 -1338.963} C_VEL
LIN {X 0,Y 587.367,Z 577.314,A -85,B 0,C 180,E1 -1341.745,E2 -1341.745} C_VEL
LIN {X 0,Y 587.361,Z 577.317,A -85,B 0,C 180,E1 -1344.507,E2 -1344.507} C_VEL
LIN {X 0,Y 587.371,Z 577.32,A -85,B 0,C 180,E1 -1347.257,E2 -1347.257} C_VEL
LIN {X 0,Y 587.382,Z 577.311,A -85,B 0,C 180,E1 -1350,E2 -1350} C_VEL
LIN {X 0,Y 587.369,Z 577.317,A -85,B 0,C 180,E1 -1352.743,E2 -1352.743} C_VEL
LIN {X 0,Y 587.364,Z 577.319,A -85,B 0,C 180,E1 -1355.493,E2 -1355.493} C_VEL
LIN {X 0,Y 587.363,Z 577.314,A -85,B 0,C 180,E1 -1358.255,E2 -1358.255} C_VEL
LIN {X 0,Y 587.345,Z 577.324,A -85,B 0,C 180,E1 -1361.133,E2 -1361.133} C_VEL
LIN {X 0,Y 587.362,Z 577.314,A -85,B 0,C 180,E1 -1364.26,E2 -1364.26} C_VEL
LIN {X 0,Y 587.356,Z 577.326,A -85,B 0,C 180,E1 -1367.405,E2 -1367.405} C_VEL
LIN {X 0,Y 587.328,Z 577.319,A -85,B 0,C 180,E1 -1370.304,E2 -1370.304} C_VEL
LIN {X 0,Y 587.319,Z 577.326,A -85,B 0,C 180,E1 -1373.258,E2 -1373.258} C_VEL
LIN {X 0,Y 587.339,Z 577.328,A -85,B 0,C 180,E1 -1375.516,E2 -1375.516} C_VEL
LIN {X 0,Y 587.37,Z 577.491,A -85,B 0,C 180,E1 -1376.803,E2 -1376.803} C_VEL
LIN {X 0,Y 587.394,Z 591.534,A -85,B 0,C 180,E1 -1379.376,E2 -1379.376} C_VEL
LIN {X 0,Y 587.31,Z 603.654,A -85,B 0,C 180,E1 -1381.568,E2 -1381.568} C_VEL
LIN {X 0,Y 587.87,Z 608.974,A -85,B 0,C 180,E1 -1381.648,E2 -1381.648} C_VEL
LIN {X 0,Y 587.736,Z 710.4,A -85,B 0,C 180,E1 -1382.908,E2 -1382.908} C_VEL
LIN {X 0,Y 587.671,Z 724.111,A -85,B 0,C 180,E1 -1383.231,E2 -1383.231} C_VEL
LIN {X 0,Y 587.613,Z 737.037,A -85,B 0,C 180,E1 -1383.686,E2 -1383.686} C_VEL
LIN {X 0,Y 587.527,Z 748.049,A -85,B 0,C 180,E1 -1384.208,E2 -1384.208} C_VEL
LIN {X 0,Y 587.427,Z 758.929,A -85,B 0,C 180,E1 -1384.862,E2 -1384.862} C_VEL
LIN {X 0,Y 587.407,Z 769.927,A -85,B 0,C 180,E1 -1385.69,E2 -1385.69} C_VEL
LIN {X 0,Y 587.32,Z 778.806,A -85,B 0,C 180,E1 -1386.512,E2 -1386.512} C_VEL
LIN {X 0,Y 587.254,Z 786.682,A -85,B 0,C 180,E1 -1387.397,E2 -1387.397} C_VEL
LIN {X 0,Y 587.226,Z 794.546,A -85,B 0,C 180,E1 -1388.486,E2 -1388.486} C_VEL
LIN {X 0,Y 587.206,Z 801.384,A -85,B 0,C 180,E1 -1389.687,E2 -1389.687} C_VEL
LIN {X 0,Y 587.165,Z 805.687,A -85,B 0,C 180,E1 -1390.66,E2 -1390.66} C_VEL
LIN {X 0,Y 587.163,Z 808.998,A -85,B 0,C 180,E1 -1391.628,E2 -1391.628} C_VEL
LIN {X 0,Y 587.158,Z 812.253,A -85,B 0,C 180,E1 -1393.019,E2 -1393.019} C_VEL
LIN {X 0,Y 587.146,Z 813.605,A -85,B 0,C 180,E1 -1394.096,E2 -1394.096} C_VEL
LIN {X 0,Y 587.133,Z 813.999,A -85,B 0,C 180,E1 -1395.072,E2 -1395.072} C_VEL
LIN {X 0,Y 587.128,Z 813.579,A -85,B 0,C 180,E1 -1396.032,E2 -1396.032} C_VEL
LIN {X 0,Y 587.158,Z 812.399,A -85,B 0,C 180,E1 -1396.98,E2 -1396.98} C_VEL
LIN {X 0,Y 587.162,Z 809.277,A -85,B 0,C 180,E1 -1398.372,E2 -1398.372} C_VEL
LIN {X 0,Y 587.159,Z 806.044,A -85,B 0,C 180,E1 -1399.339,E2 -1399.339} C_VEL
LIN {X 0,Y 587.206,Z 801.816,A -85,B 0,C 180,E1 -1400.313,E2 -1400.313} C_VEL
LIN {X 0,Y 587.228,Z 796.486,A -85,B 0,C 180,E1 -1401.294,E2 -1401.294} C_VEL
LIN {X 0,Y 587.24,Z 789.095,A -85,B 0,C 180,E1 -1402.385,E2 -1402.385} C_VEL
LIN {X 0,Y 587.271,Z 781.425,A -85,B 0,C 180,E1 -1403.301,E2 -1403.301} C_VEL
LIN {X 0,Y 587.371,Z 772.155,A -85,B 0,C 180,E1 -1404.207,E2 -1404.207} C_VEL
LIN {X 0,Y 587.437,Z 761.594,A -85,B 0,C 180,E1 -1405.045,E2 -1405.045} C_VEL
LIN {X 0,Y 587.527,Z 749.673,A -85,B 0,C 180,E1 -1405.791,E2 -1405.791} C_VEL
LIN {X 0,Y 587.594,Z 737.975,A -85,B 0,C 180,E1 -1406.364,E2 -1406.364} C_VEL
LIN {X 0,Y 587.67,Z 726.595,A -85,B 0,C 180,E1 -1406.785,E2 -1406.785} C_VEL
LIN {X 0,Y 587.702,Z 713.426,A -85,B 0,C 180,E1 -1407.124,E2 -1407.124} C_VEL
LIN {X 0,Y 587.742,Z 696.067,A -85,B 0,C 180,E1 -1407.376,E2 -1407.376} C_VEL
LIN {X 0,Y 587.711,Z 606.16,A -85,B 0,C 180,E1 -1408.48,E2 -1408.48} C_VEL
LIN {X 0,Y 587.324,Z 603.592,A -85,B 0,C 180,E1 -1408.532,E2 -1408.532} C_VEL
LIN {X 0,Y 587.416,Z 587.72,A -85,B 0,C 180,E1 -1411.408,E2 -1411.408} C_VEL
LIN {X 0,Y 587.347,Z 577.32,A -85,B 0,C 180,E1 -1413.339,E2 -1413.339} C_VEL
LIN {X 0,Y 587.331,Z 577.321,A -85,B 0,C 180,E1 -1415.994,E2 -1415.994} C_VEL
LIN {X 0,Y 587.336,Z 577.322,A -85,B 0,C 180,E1 -1418.963,E2 -1418.963} C_VEL
LIN {X 0,Y 587.325,Z 577.32,A -85,B 0,C 180,E1 -1421.874,E2 -1421.874} C_VEL
LIN {X 0,Y 587.321,Z 577.321,A -85,B 0,C 180,E1 -1424.025,E2 -1424.025} C_VEL
LIN {X 0,Y 587.353,Z 577.318,A -85,B 0,C 180,E1 -1426.155,E2 -1426.155} C_VEL
LIN {X 0,Y 587.339,Z 577.324,A -85,B 0,C 180,E1 -1428.963,E2 -1428.963} C_VEL
LIN {X 0,Y 587.366,Z 577.314,A -85,B 0,C 180,E1 -1431.745,E2 -1431.745} C_VEL
LIN {X 0,Y 587.359,Z 577.32,A -85,B 0,C 180,E1 -1434.507,E2 -1434.507} C_VEL
LIN {X 0,Y 587.378,Z 577.316,A -85,B 0,C 180,E1 -1437.257,E2 -1437.257} C_VEL
LIN {X 0,Y 587.372,Z 577.313,A -85,B 0,C 180,E1 -1440,E2 -1440} C_VEL
LIN {X 0,Y 587.377,Z 577.32,A -85,B 0,C 180,E1 -1442.744,E2 -1442.744} C_VEL
LIN {X 0,Y 587.361,Z 577.317,A -85,B 0,C 180,E1 -1445.493,E2 -1445.493} C_VEL
LIN {X 0,Y 587.365,Z 577.315,A -85,B 0,C 180,E1 -1448.256,E2 -1448.256} C_VEL
LIN {X 0,Y 587.352,Z 577.324,A -85,B 0,C 180,E1 -1451.142,E2 -1451.142} C_VEL
LIN {X 0,Y 587.355,Z 577.316,A -85,B 0,C 180,E1 -1454.262,E2 -1454.262} C_VEL
LIN {X 0,Y 587.353,Z 577.321,A -85,B 0,C 180,E1 -1457.406,E2 -1457.406} C_VEL
LIN {X 0,Y 587.326,Z 577.319,A -85,B 0,C 180,E1 -1460.305,E2 -1460.305} C_VEL
LIN {X 0,Y 587.317,Z 577.329,A -85,B 0,C 180,E1 -1463.259,E2 -1463.259} C_VEL
LIN {X 0,Y 587.355,Z 577.315,A -85,B 0,C 180,E1 -1466.183,E2 -1466.183} C_VEL
LIN {X 0,Y 587.344,Z 577.325,A -85,B 0,C 180,E1 -1469.135,E2 -1469.135} C_VEL
LIN {X 0,Y 587.349,Z 577.317,A -85,B 0,C 180,E1 -1471.839,E2 -1471.839} C_VEL
LIN {X 0,Y 587.35,Z 577.315,A -85,B 0,C 180,E1 -1474.35,E2 -1474.35} C_VEL
LIN {X 0,Y 587.348,Z 577.318,A -85,B 0,C 180,E1 -1476.747,E2 -1476.747} C_VEL
LIN {X 0,Y 587.344,Z 577.327,A -85,B 0,C 180,E1 -1479.36,E2 -1479.36} C_VEL
LIN {X 0,Y 587.33,Z 577.32,A -85,B 0,C 180,E1 -1482.109,E2 -1482.109} C_VEL
LIN {X 0,Y 587.312,Z 577.325,A -85,B 0,C 180,E1 -1485.09,E2 -1485.09} C_VEL
LIN {X 0,Y 587.35,Z 577.32,A -85,B 0,C 180,E1 -1487.929,E2 -1487.929} C_VEL
LIN {X 0,Y 587.331,Z 577.321,A -85,B 0,C 180,E1 -1491.059,E2 -1491.059} C_VEL
LIN {X 0,Y 587.352,Z 577.322,A -85,B 0,C 180,E1 -1493.293,E2 -1493.293} C_VEL
LIN {X 0,Y 587.366,Z 577.322,A -85,B 0,C 180,E1 -1495.781,E2 -1495.781} C_VEL
LIN {X 0,Y 587.343,Z 577.318,A -85,B 0,C 180,E1 -1498.232,E2 -1498.232} C_VEL
LIN {X 0,Y 587.35,Z 577.317,A -85,B 0,C 180,E1 -1500.867,E2 -1500.867} C_VEL
LIN {X 0,Y 587.36,Z 577.325,A -85,B 0,C 180,E1 -1503.82,E2 -1503.82} C_VEL
LIN {X 0,Y 587.386,Z 577.484,A -85,B 0,C 180,E1 -1506.418,E2 -1506.418} C_VEL
LIN {X 0,Y 587.894,Z 581.48,A -85,B 0,C 180,E1 -1507,E2 -1507} C_VEL
LIN {X 0,Y 587.767,Z 601.083,A -85,B 0,C 180,E1 -1509.712,E2 -1509.712} C_VEL
LIN {X 0,Y 587.597,Z 622.357,A -85,B 0,C 180,E1 -1512.602,E2 -1512.602} C_VEL
LIN {X 0,Y 587.478,Z 643.63,A -85,B 0,C 180,E1 -1515.45,E2 -1515.45} C_VEL
LIN {X 0,Y 587.432,Z 651.524,A -85,B 0,C 180,E1 -1516.498,E2 -1516.498} C_VEL
LIN {X 0,Y 587.87,Z 655.747,A -85,B 0,C 180,E1 -1516.563,E2 -1516.563} C_VEL
LIN {X 0,Y 587.742,Z 759.963,A -85,B 0,C 180,E1 -1517.856,E2 -1517.856} C_VEL
LIN {X 0,Y 587.703,Z 772.469,A -85,B 0,C 180,E1 -1518.139,E2 -1518.139} C_VEL
LIN {X 0,Y 587.632,Z 784.592,A -85,B 0,C 180,E1 -1518.545,E2 -1518.545} C_VEL
LIN {X 0,Y 587.542,Z 795.931,A -85,B 0,C 180,E1 -1519.054,E2 -1519.054} C_VEL
LIN {X 0,Y 587.471,Z 806.586,A -85,B 0,C 180,E1 -1519.663,E2 -1519.663} C_VEL
LIN {X 0,Y 587.39,Z 817.479,A -85,B 0,C 180,E1 -1520.444,E2 -1520.444} C_VEL
LIN {X 0,Y 587.321,Z 828.114,A -85,B 0,C 180,E1 -1521.398,E2 -1521.398} C_VEL
LIN {X 0,Y 587.274,Z 835.962,A -85,B 0,C 180,E1 -1522.263,E2 -1522.263} C_VEL
LIN {X 0,Y 587.23,Z 842.471,A -85,B 0,C 180,E1 -1523.127,E2 -1523.127} C_VEL
LIN {X 0,Y 587.236,Z 848.867,A -85,B 0,C 180,E1 -1524.161,E2 -1524.161} C_VEL
LIN {X 0,Y 587.147,Z 853.95,A -85,B 0,C 180,E1 -1525.194,E2 -1525.194} C_VEL
LIN {X 0,Y 587.213,Z 857.896,A -85,B 0,C 180,E1 -1526.226,E2 -1526.226} C_VEL
LIN {X 0,Y 587.132,Z 860.809,A -85,B 0,C 180,E1 -1527.256,E2 -1527.256} C_VEL
LIN {X 0,Y 587.138,Z 862.201,A -85,B 0,C 180,E1 -1527.942,E2 -1527.942} C_VEL
LIN {X 0,Y 587.14,Z 863.784,A -85,B 0,C 180,E1 -1529.314,E2 -1529.314} C_VEL
LIN {X 0,Y 587.137,Z 864,A -85,B 0,C 180,E1 -1530,E2 -1530} C_VEL
LIN {X 0,Y 587.147,Z 863.185,A -85,B 0,C 180,E1 -1531.372,E2 -1531.372} C_VEL
LIN {X 0,Y 587.138,Z 862.201,A -85,B 0,C 180,E1 -1532.058,E2 -1532.058} C_VEL
LIN {X 0,Y 587.132,Z 860.81,A -85,B 0,C 180,E1 -1532.744,E2 -1532.744} C_VEL
LIN {X 0,Y 587.213,Z 857.896,A -85,B 0,C 180,E1 -1533.774,E2 -1533.774} C_VEL
LIN {X 0,Y 587.147,Z 853.95,A -85,B 0,C 180,E1 -1534.806,E2 -1534.806} C_VEL
LIN {X 0,Y 587.217,Z 847.878,A -85,B 0,C 180,E1 -1536.011,E2 -1536.011} C_VEL
LIN {X 0,Y 587.245,Z 841.238,A -85,B 0,C 180,E1 -1537.046,E2 -1537.046} C_VEL
LIN {X 0,Y 587.299,Z 832.992,A -85,B 0,C 180,E1 -1538.083,E2 -1538.083} C_VEL
LIN {X 0,Y 587.343,Z 824.54,A -85,B 0,C 180,E1 -1538.949,E2 -1538.949} C_VEL
LIN {X 0,Y 587.411,Z 814.098,A -85,B 0,C 180,E1 -1539.816,E2 -1539.816} C_VEL
LIN {X 0,Y 587.507,Z 803.763,A -85,B 0,C 180,E1 -1540.511,E2 -1540.511} C_VEL
LIN {X 0,Y 587.583,Z 791.81,A -85,B 0,C 180,E1 -1541.149,E2 -1541.149} C_VEL
LIN {X 0,Y 587.657,Z 779.601,A -85,B 0,C 180,E1 -1541.639,E2 -1541.639} C_VEL
LIN {X 0,Y 587.678,Z 766.449,A -85,B 0,C 180,E1 -1542.014,E2 -1542.014} C_VEL
LIN {X 0,Y 587.744,Z 754.107,A -85,B 0,C 180,E1 -1542.232,E2 -1542.232} C_VEL
LIN {X 0,Y 587.733,Z 653.511,A -85,B 0,C 180,E1 -1543.467,E2 -1543.467} C_VEL
LIN {X 0,Y 587.42,Z 651.441,A -85,B 0,C 180,E1 -1543.513,E2 -1543.513} C_VEL
LIN {X 0,Y 587.553,Z 629.005,A -85,B 0,C 180,E1 -1546.504,E2 -1546.504} C_VEL
LIN {X 0,Y 587.68,Z 609.545,A -85,B 0,C 180,E1 -1549.134,E2 -1549.134} C_VEL
LIN {X 0,Y 587.871,Z 589.117,A -85,B 0,C 180,E1 -1551.937,E2 -1551.937} C_VEL
LIN {X 0,Y 587.824,Z 579.81,A -85,B 0,C 180,E1 -1553.237,E2 -1553.237} C_VEL
LIN {X 0,Y 587.345,Z 577.324,A -85,B 0,C 180,E1 -1553.631,E2 -1553.631} C_VEL
LIN {X 0,Y 587.34,Z 577.328,A -85,B 0,C 180,E1 -1556.278,E2 -1556.278} C_VEL
LIN {X 0,Y 587.35,Z 577.317,A -85,B 0,C 180,E1 -1559.133,E2 -1559.133} C_VEL
LIN {X 0,Y 587.346,Z 577.319,A -85,B 0,C 180,E1 -1561.835,E2 -1561.835} C_VEL
LIN {X 0,Y 587.354,Z 577.324,A -85,B 0,C 180,E1 -1564.348,E2 -1564.348} C_VEL
LIN {X 0,Y 587.351,Z 577.322,A -85,B 0,C 180,E1 -1566.746,E2 -1566.746} C_VEL
LIN {X 0,Y 587.343,Z 577.317,A -85,B 0,C 180,E1 -1569.358,E2 -1569.358} C_VEL
LIN {X 0,Y 587.331,Z 577.321,A -85,B 0,C 180,E1 -1572.107,E2 -1572.107} C_VEL
LIN {X 0,Y 587.312,Z 577.324,A -85,B 0,C 180,E1 -1575.088,E2 -1575.088} C_VEL
LIN {X 0,Y 587.348,Z 577.316,A -85,B 0,C 180,E1 -1577.927,E2 -1577.927} C_VEL
LIN {X 0,Y 587.331,Z 577.323,A -85,B 0,C 180,E1 -1581.057,E2 -1581.057} C_VEL
LIN {X 0,Y 587.349,Z 577.318,A -85,B 0,C 180,E1 -1583.291,E2 -1583.291} C_VEL
LIN {X 0,Y 587.36,Z 577.314,A -85,B 0,C 180,E1 -1585.78,E2 -1585.78} C_VEL
LIN {X 0,Y 587.346,Z 577.317,A -85,B 0,C 180,E1 -1588.231,E2 -1588.231} C_VEL
LIN {X 0,Y 587.344,Z 577.326,A -85,B 0,C 180,E1 -1590.865,E2 -1590.865} C_VEL
LIN {X 0,Y 587.354,Z 577.315,A -85,B 0,C 180,E1 -1593.817,E2 -1593.817} C_VEL
LIN {X 0,Y 587.331,Z 577.318,A -85,B 0,C 180,E1 -1595.993,E2 -1595.993} C_VEL
LIN {X 0,Y 587.339,Z 577.326,A -85,B 0,C 180,E1 -1598.962,E2 -1598.962} C_VEL
LIN {X 0,Y 587.321,Z 577.32,A -85,B 0,C 180,E1 -1601.873,E2 -1601.873} C_VEL
LIN {X 0,Y 587.318,Z 577.32,A -85,B 0,C 180,E1 -1604.024,E2 -1604.024} C_VEL
LIN {X 0,Y 587.351,Z 577.315,A -85,B 0,C 180,E1 -1606.154,E2 -1606.154} C_VEL
LIN {X 0,Y 587.338,Z 577.323,A -85,B 0,C 180,E1 -1608.962,E2 -1608.962} C_VEL
LIN {X 0,Y 587.365,Z 577.317,A -85,B 0,C 180,E1 -1611.744,E2 -1611.744} C_VEL
LIN {X 0,Y 587.355,Z 577.315,A -85,B 0,C 180,E1 -1614.507,E2 -1614.507} C_VEL
LIN {X 0,Y 587.375,Z 577.321,A -85,B 0,C 180,E1 -1617.256,E2 -1617.256} C_VEL
LIN {X 0,Y 587.372,Z 577.315,A -85,B 0,C 180,E1 -1620,E2 -1620} C_VEL
LIN {X 0,Y 587.375,Z 577.313,A -85,B 0,C 180,E1 -1622.743,E2 -1622.743} C_VEL
LIN {X 0,Y 587.35,Z 577.326,A -85,B 0,C 180,E1 -1625.493,E2 -1625.493} C_VEL
LIN {X 0,Y 587.364,Z 577.315,A -85,B 0,C 180,E1 -1628.255,E2 -1628.255} C_VEL
LIN {X 0,Y 587.35,Z 577.318,A -85,B 0,C 180,E1 -1631.141,E2 -1631.141} C_VEL
LIN {X 0,Y 587.353,Z 577.317,A -85,B 0,C 180,E1 -1634.261,E2 -1634.261} C_VEL
LIN {X 0,Y 587.349,Z 577.32,A -85,B 0,C 180,E1 -1637.406,E2 -1637.406} C_VEL
LIN {X 0,Y 587.317,Z 577.322,A -85,B 0,C 180,E1 -1638.324,E2 -1638.324} C_VEL
LIN {X 0,Y 586.664,Z 577.403,A -85,B 0,C 180,E1 -1638.896,E2 -1638.896} C_VEL
LIN {X 0,Y 583.832,Z 577.765,A -85,B 0,C 180,E1 -1639.825,E2 -1639.825} C_VEL
LIN {X 0,Y 581.423,Z 578.061,A -85,B 0,C 180,E1 -1640.572,E2 -1640.572} C_VEL
LIN {X 0,Y 580.371,Z 578.188,A -85,B 0,C 180,E1 -1641.148,E2 -1641.148} C_VEL
LIN {X 0,Y 580.276,Z 578.199,A -85,B 0,C 180,E1 -1641.343,E2 -1641.343} C_VEL
LIN {X 0,Y 580.291,Z 578.199,A -85,B 0,C 180,E1 -1644.316,E2 -1644.316} C_VEL
LIN {X 0,Y 580.3,Z 578.195,A -85,B 0,C 180,E1 -1646.622,E2 -1646.622} C_VEL
LIN {X 0,Y 580.296,Z 578.195,A -85,B 0,C 180,E1 -1649.311,E2 -1649.311} C_VEL
LIN {X 0,Y 580.293,Z 578.203,A -85,B 0,C 180,E1 -1652.2,E2 -1652.2} C_VEL
LIN {X 0,Y 580.29,Z 578.197,A -85,B 0,C 180,E1 -1654.696,E2 -1654.696} C_VEL
LIN {X 0,Y 580.293,Z 578.195,A -85,B 0,C 180,E1 -1657.268,E2 -1657.268} C_VEL
LIN {X 0,Y 580.298,Z 578.203,A -85,B 0,C 180,E1 -1660.273,E2 -1660.273} C_VEL
LIN {X 0,Y 580.29,Z 578.198,A -85,B 0,C 180,E1 -1662.705,E2 -1662.705} C_VEL
LIN {X 0,Y 580.265,Z 578.199,A -85,B 0,C 180,E1 -1665.609,E2 -1665.609} C_VEL
LIN {X 0,Y 580.306,Z 578.202,A -85,B 0,C 180,E1 -1668.235,E2 -1668.235} C_VEL
LIN {X 0,Y 580.282,Z 578.198,A -85,B 0,C 180,E1 -1670.967,E2 -1670.967} C_VEL
LIN {X 0,Y 580.29,Z 578.195,A -85,B 0,C 180,E1 -1673.599,E2 -1673.599} C_VEL
LIN {X 0,Y 580.316,Z 578.197,A -85,B 0,C 180,E1 -1676.146,E2 -1676.146} C_VEL
LIN {X 0,Y 580.284,Z 578.205,A -85,B 0,C 180,E1 -1678.616,E2 -1678.616} C_VEL
LIN {X 0,Y 580.29,Z 578.198,A -85,B 0,C 180,E1 -1681.025,E2 -1681.025} C_VEL
LIN {X 0,Y 580.287,Z 578.195,A -85,B 0,C 180,E1 -1683.666,E2 -1683.666} C_VEL
LIN {X 0,Y 580.296,Z 578.194,A -85,B 0,C 180,E1 -1685.684,E2 -1685.684} C_VEL
LIN {X 0,Y 580.271,Z 578.198,A -85,B 0,C 180,E1 -1687.948,E2 -1687.948} C_VEL
LIN {X 0,Y 580.315,Z 578.2,A -85,B 0,C 180,E1 -1690.914,E2 -1690.914} C_VEL
LIN {X 0,Y 580.278,Z 578.196,A -85,B 0,C 180,E1 -1693.826,E2 -1693.826} C_VEL
LIN {X 0,Y 580.324,Z 578.191,A -85,B 0,C 180,E1 -1695.983,E2 -1695.983} C_VEL
LIN {X 0,Y 580.301,Z 578.204,A -85,B 0,C 180,E1 -1698.827,E2 -1698.827} C_VEL
LIN {X 0,Y 580.331,Z 578.191,A -85,B 0,C 180,E1 -1701.644,E2 -1701.644} C_VEL
LIN {X 0,Y 580.327,Z 578.193,A -85,B 0,C 180,E1 -1704.44,E2 -1704.44} C_VEL
LIN {X 0,Y 580.337,Z 578.196,A -85,B 0,C 180,E1 -1707.224,E2 -1707.224} C_VEL
LIN {X 0,Y 580.352,Z 578.187,A -85,B 0,C 180,E1 -1710,E2 -1710} C_VEL
LIN {X 0,Y 580.336,Z 578.194,A -85,B 0,C 180,E1 -1712.776,E2 -1712.776} C_VEL
LIN {X 0,Y 580.33,Z 578.194,A -85,B 0,C 180,E1 -1715.56,E2 -1715.56} C_VEL
LIN {X 0,Y 580.326,Z 578.191,A -85,B 0,C 180,E1 -1718.356,E2 -1718.356} C_VEL
LIN {X 0,Y 580.297,Z 578.203,A -85,B 0,C 180,E1 -1721.191,E2 -1721.191} C_VEL
LIN {X 0,Y 580.325,Z 578.192,A -85,B 0,C 180,E1 -1724.017,E2 -1724.017} C_VEL
LIN {X 0,Y 580.309,Z 578.196,A -85,B 0,C 180,E1 -1726.914,E2 -1726.914} C_VEL
LIN {X 0,Y 580.303,Z 578.198,A -85,B 0,C 180,E1 -1729.822,E2 -1729.822} C_VEL
LIN {X 0,Y 580.291,Z 578.196,A -85,B 0,C 180,E1 -1732.802,E2 -1732.802} C_VEL
LIN {X 0,Y 580.306,Z 578.198,A -85,B 0,C 180,E1 -1735.079,E2 -1735.079} C_VEL
LIN {X 0,Y 580.319,Z 578.262,A -85,B 0,C 180,E1 -1736.718,E2 -1736.718} C_VEL
LIN {X 0,Y 580.373,Z 590.391,A -85,B 0,C 180,E1 -1738.971,E2 -1738.971} C_VEL
LIN {X 0,Y 580.274,Z 603.56,A -85,B 0,C 180,E1 -1741.385,E2 -1741.385} C_VEL
LIN {X 0,Y 580.97,Z 608.696,A -85,B 0,C 180,E1 -1741.482,E2 -1741.482} C_VEL
LIN {X 0,Y 580.802,Z 710.286,A -85,B 0,C 180,E1 -1742.759,E2 -1742.759} C_VEL
LIN {X 0,Y 580.726,Z 723.864,A -85,B 0,C 180,E1 -1743.08,E2 -1743.08} C_VEL
LIN {X 0,Y 580.645,Z 736.288,A -85,B 0,C 180,E1 -1743.518,E2 -1743.518} C_VEL
LIN {X 0,Y 580.539,Z 747.544,A -85,B 0,C 180,E1 -1744.048,E2 -1744.048} C_VEL
LIN {X 0,Y 580.43,Z 758.164,A -85,B 0,C 180,E1 -1744.686,E2 -1744.686} C_VEL
LIN {X 0,Y 580.356,Z 769.484,A -85,B 0,C 180,E1 -1745.539,E2 -1745.539} C_VEL
LIN {X 0,Y 580.28,Z 778.751,A -85,B 0,C 180,E1 -1746.402,E2 -1746.402} C_VEL
LIN {X 0,Y 580.188,Z 787.979,A -85,B 0,C 180,E1 -1747.47,E2 -1747.47} C_VEL
LIN {X 0,Y 580.164,Z 795.762,A -85,B 0,C 180,E1 -1748.597,E2 -1748.597} C_VEL
LIN {X 0,Y 580.133,Z 800.912,A -85,B 0,C 180,E1 -1749.528,E2 -1749.528} C_VEL
LIN {X 0,Y 580.099,Z 805.378,A -85,B 0,C 180,E1 -1750.53,E2 -1750.53} C_VEL
LIN {X 0,Y 580.095,Z 809.58,A -85,B 0,C 180,E1 -1751.784,E2 -1751.784} C_VEL
LIN {X 0,Y 580.063,Z 811.767,A -85,B 0,C 180,E1 -1752.725,E2 -1752.725} C_VEL
LIN {X 0,Y 580.019,Z 813.213,A -85,B 0,C 180,E1 -1753.681,E2 -1753.681} C_VEL
LIN {X 0,Y 580.025,Z 813.917,A -85,B 0,C 180,E1 -1754.648,E2 -1754.648} C_VEL
LIN {X 0,Y 580.029,Z 813.856,A -85,B 0,C 180,E1 -1755.632,E2 -1755.632} C_VEL
LIN {X 0,Y 580.024,Z 812.956,A -85,B 0,C 180,E1 -1756.634,E2 -1756.634} C_VEL
LIN {X 0,Y 580.072,Z 811.18,A -85,B 0,C 180,E1 -1757.65,E2 -1757.65} C_VEL
LIN {X 0,Y 580.059,Z 808.426,A -85,B 0,C 180,E1 -1758.692,E2 -1758.692} C_VEL
LIN {X 0,Y 580.114,Z 804.609,A -85,B 0,C 180,E1 -1759.749,E2 -1759.749} C_VEL
LIN {X 0,Y 580.133,Z 798.875,A -85,B 0,C 180,E1 -1760.954,E2 -1760.954} C_VEL
LIN {X 0,Y 580.166,Z 791.535,A -85,B 0,C 180,E1 -1762.136,E2 -1762.136} C_VEL
LIN {X 0,Y 580.236,Z 783.183,A -85,B 0,C 180,E1 -1763.205,E2 -1763.205} C_VEL
LIN {X 0,Y 580.332,Z 774.385,A -85,B 0,C 180,E1 -1764.116,E2 -1764.116} C_VEL
LIN {X 0,Y 580.411,Z 763.9,A -85,B 0,C 180,E1 -1764.996,E2 -1764.996} C_VEL
LIN {X 0,Y 580.491,Z 752.893,A -85,B 0,C 180,E1 -1765.739,E2 -1765.739} C_VEL
LIN {X 0,Y 580.614,Z 740.97,A -85,B 0,C 180,E1 -1766.367,E2 -1766.367} C_VEL
LIN {X 0,Y 580.697,Z 728.358,A -85,B 0,C 180,E1 -1766.868,E2 -1766.868} C_VEL
LIN {X 0,Y 580.758,Z 715.633,A -85,B 0,C 180,E1 -1767.225,E2 -1767.225} C_VEL
LIN {X 0,Y 580.819,Z 701.266,A -85,B 0,C 180,E1 -1767.46,E2 -1767.46} C_VEL
LIN {X 0,Y 580.879,Z 607.392,A -85,B 0,C 180,E1 -1768.626,E2 -1768.626} C_VEL
LIN {X 0,Y 580.276,Z 603.542,A -85,B 0,C 180,E1 -1768.709,E2 -1768.709} C_VEL
LIN {X 0,Y 580.382,Z 588.733,A -85,B 0,C 180,E1 -1771.425,E2 -1771.425} C_VEL
LIN {X 0,Y 580.332,Z 578.22,A -85,B 0,C 180,E1 -1773.38,E2 -1773.38} C_VEL
LIN {X 0,Y 580.292,Z 578.197,A -85,B 0,C 180,E1 -1775.684,E2 -1775.684} C_VEL
LIN {X 0,Y 580.267,Z 578.2,A -85,B 0,C 180,E1 -1777.948,E2 -1777.948} C_VEL
LIN {X 0,Y 580.306,Z 578.199,A -85,B 0,C 180,E1 -1780.914,E2 -1780.914} C_VEL
LIN {X 0,Y 580.274,Z 578.198,A -85,B 0,C 180,E1 -1783.826,E2 -1783.826} C_VEL
LIN {X 0,Y 580.276,Z 578.208,A -85,B 0,C 180,E1 -1786.696,E2 -1786.696} C_VEL
LIN {X 0,Y 580.299,Z 578.195,A -85,B 0,C 180,E1 -1789.534,E2 -1789.534} C_VEL
LIN {X 0,Y 580.332,Z 578.194,A -85,B 0,C 180,E1 -1792.345,E2 -1792.345} C_VEL
LIN {X 0,Y 580.339,Z 578.194,A -85,B 0,C 180,E1 -1795.138,E2 -1795.138} C_VEL
LIN {X 0,Y 580.329,Z 578.191,A -85,B 0,C 180,E1 -1797.918,E2 -1797.918} C_VEL
LIN {X 0,Y 580.36,Z 578.194,A -85,B 0,C 180,E1 -1800.694,E2 -1800.694} C_VEL
LIN {X 0,Y 580.284,Z 578.198,A -85,B 0,C 180,E1 -1803.472,E2 -1803.472} C_VEL
LIN {X 0,Y 580.327,Z 578.192,A -85,B 0,C 180,E1 -1805.56,E2 -1805.56} C_VEL
LIN {X 0,Y 580.329,Z 578.192,A -85,B 0,C 180,E1 -1808.356,E2 -1808.356} C_VEL
LIN {X 0,Y 580.323,Z 578.198,A -85,B 0,C 180,E1 -1811.209,E2 -1811.209} C_VEL
LIN {X 0,Y 580.318,Z 578.192,A -85,B 0,C 180,E1 -1814.017,E2 -1814.017} C_VEL
LIN {X 0,Y 580.303,Z 578.2,A -85,B 0,C 180,E1 -1816.915,E2 -1816.915} C_VEL
LIN {X 0,Y 580.3,Z 578.195,A -85,B 0,C 180,E1 -1819.823,E2 -1819.823} C_VEL
LIN {X 0,Y 580.267,Z 578.198,A -85,B 0,C 180,E1 -1822.053,E2 -1822.053} C_VEL
LIN {X 0,Y 580.302,Z 578.202,A -85,B 0,C 180,E1 -1825.08,E2 -1825.08} C_VEL
LIN {X 0,Y 580.312,Z 578.194,A -85,B 0,C 180,E1 -1827.864,E2 -1827.864} C_VEL
LIN {X 0,Y 580.293,Z 578.196,A -85,B 0,C 180,E1 -1830.698,E2 -1830.698} C_VEL
LIN {X 0,Y 580.3,Z 578.205,A -85,B 0,C 180,E1 -1833.318,E2 -1833.318} C_VEL
LIN {X 0,Y 580.32,Z 578.195,A -85,B 0,C 180,E1 -1835.768,E2 -1835.768} C_VEL
LIN {X 0,Y 580.286,Z 578.196,A -85,B 0,C 180,E1 -1838.147,E2 -1838.147} C_VEL
LIN {X 0,Y 580.297,Z 578.196,A -85,B 0,C 180,E1 -1840.844,E2 -1840.844} C_VEL
LIN {X 0,Y 580.284,Z 578.203,A -85,B 0,C 180,E1 -1843.658,E2 -1843.658} C_VEL
LIN {X 0,Y 580.273,Z 578.198,A -85,B 0,C 180,E1 -1846.61,E2 -1846.61} C_VEL
LIN {X 0,Y 580.296,Z 578.199,A -85,B 0,C 180,E1 -1849.158,E2 -1849.158} C_VEL
LIN {X 0,Y 580.288,Z 578.2,A -85,B 0,C 180,E1 -1851.928,E2 -1851.928} C_VEL
LIN {X 0,Y 580.306,Z 578.194,A -85,B 0,C 180,E1 -1854.458,E2 -1854.458} C_VEL
LIN {X 0,Y 580.292,Z 578.197,A -85,B 0,C 180,E1 -1856.976,E2 -1856.976} C_VEL
LIN {X 0,Y 580.294,Z 578.201,A -85,B 0,C 180,E1 -1859.426,E2 -1859.426} C_VEL
LIN {X 0,Y 580.298,Z 578.199,A -85,B 0,C 180,E1 -1862.142,E2 -1862.142} C_VEL
LIN {X 0,Y 580.322,Z 578.197,A -85,B 0,C 180,E1 -1865.27,E2 -1865.27} C_VEL
LIN {X 0,Y 580.311,Z 578.315,A -85,B 0,C 180,E1 -1866.231,E2 -1866.231} C_VEL
LIN {X 0,Y 580.998,Z 583.185,A -85,B 0,C 180,E1 -1866.952,E2 -1866.952} C_VEL
LIN {X 0,Y 580.843,Z 602.413,A -85,B 0,C 180,E1 -1869.644,E2 -1869.644} C_VEL
LIN {X 0,Y 580.606,Z 623.819,A -85,B 0,C 180,E1 -1872.586,E2 -1872.586} C_VEL
LIN {X 0,Y 580.454,Z 645.41,A -85,B 0,C 180,E1 -1875.51,E2 -1875.51} C_VEL
LIN {X 0,Y 580.41,Z 651.524,A -85,B 0,C 180,E1 -1876.332,E2 -1876.332} C_VEL
LIN {X 0,Y 580.983,Z 655.747,A -85,B 0,C 180,E1 -1876.401,E2 -1876.401} C_VEL
LIN {X 0,Y 580.823,Z 759.963,A -85,B 0,C 180,E1 -1877.709,E2 -1877.709} C_VEL
LIN {X 0,Y 580.75,Z 772.468,A -85,B 0,C 180,E1 -1877.995,E2 -1877.995} C_VEL
LIN {X 0,Y 580.673,Z 785.379,A -85,B 0,C 180,E1 -1878.437,E2 -1878.437} C_VEL
LIN {X 0,Y 580.563,Z 797.636,A -85,B 0,C 180,E1 -1879.009,E2 -1879.009} C_VEL
LIN {X 0,Y 580.431,Z 809.206,A -85,B 0,C 180,E1 -1879.712,E2 -1879.712} C_VEL
LIN {X 0,Y 580.341,Z 819.601,A -85,B 0,C 180,E1 -1880.503,E2 -1880.503} C_VEL
LIN {X 0,Y 580.271,Z 828.114,A -85,B 0,C 180,E1 -1881.292,E2 -1881.292} C_VEL
LIN {X 0,Y 580.222,Z 835.962,A -85,B 0,C 180,E1 -1882.168,E2 -1882.168} C_VEL
LIN {X 0,Y 580.154,Z 843.651,A -85,B 0,C 180,E1 -1883.222,E2 -1883.222} C_VEL
LIN {X 0,Y 580.139,Z 850.681,A -85,B 0,C 180,E1 -1884.439,E2 -1884.439} C_VEL
LIN {X 0,Y 580.108,Z 855.372,A -85,B 0,C 180,E1 -1885.484,E2 -1885.484} C_VEL
LIN {X 0,Y 580.123,Z 858.957,A -85,B 0,C 180,E1 -1886.527,E2 -1886.527} C_VEL
LIN {X 0,Y 580.043,Z 860.809,A -85,B 0,C 180,E1 -1887.222,E2 -1887.222} C_VEL
LIN {X 0,Y 580.038,Z 862.2,A -85,B 0,C 180,E1 -1887.917,E2 -1887.917} C_VEL
LIN {X 0,Y 580.04,Z 863.784,A -85,B 0,C 180,E1 -1889.306,E2 -1889.306} C_VEL
LIN {X 0,Y 580.037,Z 864,A -85,B 0,C 180,E1 -1890,E2 -1890} C_VEL
LIN {X 0,Y 580.047,Z 863.185,A -85,B 0,C 180,E1 -1891.389,E2 -1891.389} C_VEL
LIN {X 0,Y 580.038,Z 862.201,A -85,B 0,C 180,E1 -1892.083,E2 -1892.083} C_VEL
LIN {X 0,Y 580.043,Z 860.81,A -85,B 0,C 180,E1 -1892.778,E2 -1892.778} C_VEL
LIN {X 0,Y 580.11,Z 857.896,A -85,B 0,C 180,E1 -1893.82,E2 -1893.82} C_VEL
LIN {X 0,Y 580.054,Z 853.95,A -85,B 0,C 180,E1 -1894.865,E2 -1894.865} C_VEL
LIN {X 0,Y 580.139,Z 847.878,A -85,B 0,C 180,E1 -1896.085,E2 -1896.085} C_VEL
LIN {X 0,Y 580.184,Z 841.238,A -85,B 0,C 180,E1 -1897.132,E2 -1897.132} C_VEL
LIN {X 0,Y 580.25,Z 832.992,A -85,B 0,C 180,E1 -1898.182,E2 -1898.182} C_VEL
LIN {X 0,Y 580.308,Z 824.54,A -85,B 0,C 180,E1 -1899.058,E2 -1899.058} C_VEL
LIN {X 0,Y 580.417,Z 814.099,A -85,B 0,C 180,E1 -1899.936,E2 -1899.936} C_VEL
LIN {X 0,Y 580.512,Z 803.762,A -85,B 0,C 180,E1 -1900.639,E2 -1900.639} C_VEL
LIN {X 0,Y 580.597,Z 792.242,A -85,B 0,C 180,E1 -1901.264,E2 -1901.264} C_VEL
LIN {X 0,Y 580.707,Z 779.48,A -85,B 0,C 180,E1 -1901.784,E2 -1901.784} C_VEL
LIN {X 0,Y 580.735,Z 766.448,A -85,B 0,C 180,E1 -1902.16,E2 -1902.16} C_VEL
LIN {X 0,Y 580.83,Z 754.107,A -85,B 0,C 180,E1 -1902.38,E2 -1902.38} C_VEL
LIN {X 0,Y 580.819,Z 654.184,A -85,B 0,C 180,E1 -1903.622,E2 -1903.622} C_VEL
LIN {X 0,Y 580.425,Z 651.441,A -85,B 0,C 180,E1 -1903.679,E2 -1903.679} C_VEL
LIN {X 0,Y 580.599,Z 627.675,A -85,B 0,C 180,E1 -1906.888,E2 -1906.888} C_VEL
LIN {X 0,Y 580.785,Z 606.402,A -85,B 0,C 180,E1 -1909.805,E2 -1909.805} C_VEL
LIN {X 0,Y 581.03,Z 585.129,A -85,B 0,C 180,E1 -1912.771,E2 -1912.771} C_VEL
LIN {X 0,Y 580.949,Z 581.499,A -85,B 0,C 180,E1 -1913.289,E2 -1913.289} C_VEL
LIN {X 0,Y 580.301,Z 578.203,A -85,B 0,C 180,E1 -1913.793,E2 -1913.793} C_VEL
LIN {X 0,Y 580.278,Z 578.203,A -85,B 0,C 180,E1 -1916.623,E2 -1916.623} C_VEL
LIN {X 0,Y 580.302,Z 578.194,A -85,B 0,C 180,E1 -1919.309,E2 -1919.309} C_VEL
LIN {X 0,Y 580.3,Z 578.201,A -85,B 0,C 180,E1 -1922.2,E2 -1922.2} C_VEL
LIN {X 0,Y 580.3,Z 578.2,A -85,B 0,C 180,E1 -1924.695,E2 -1924.695} C_VEL
LIN {X 0,Y 580.297,Z 578.195,A -85,B 0,C 180,E1 -1927.267,E2 -1927.267} C_VEL
LIN {X 0,Y 580.295,Z 578.2,A -85,B 0,C 180,E1 -1930.27,E2 -1930.27} C_VEL
LIN {X 0,Y 580.274,Z 578.206,A -85,B 0,C 180,E1 -1932.705,E2 -1932.705} C_VEL
LIN {X 0,Y 580.27,Z 578.197,A -85,B 0,C 180,E1 -1935.608,E2 -1935.608} C_VEL
LIN {X 0,Y 580.31,Z 578.196,A -85,B 0,C 180,E1 -1938.233,E2 -1938.233} C_VEL
LIN {X 0,Y 580.287,Z 578.202,A -85,B 0,C 180,E1 -1940.965,E2 -1940.965} C_VEL
LIN {X 0,Y 580.291,Z 578.195,A -85,B 0,C 180,E1 -1943.598,E2 -1943.598} C_VEL
LIN {X 0,Y 580.313,Z 578.193,A -85,B 0,C 180,E1 -1946.145,E2 -1946.145} C_VEL
LIN {X 0,Y 580.284,Z 578.202,A -85,B 0,C 180,E1 -1948.615,E2 -1948.615} C_VEL
LIN {X 0,Y 580.287,Z 578.205,A -85,B 0,C 180,E1 -1951.023,E2 -1951.023} C_VEL
LIN {X 0,Y 580.32,Z 578.192,A -85,B 0,C 180,E1 -1953.658,E2 -1953.658} C_VEL
LIN {X 0,Y 580.273,Z 578.199,A -85,B 0,C 180,E1 -1956.441,E2 -1956.441} C_VEL
LIN {X 0,Y 580.274,Z 578.202,A -85,B 0,C 180,E1 -1959.437,E2 -1959.437} C_VEL
LIN {X 0,Y 580.273,Z 578.2,A -85,B 0,C 180,E1 -1961.645,E2 -1961.645} C_VEL
LIN {X 0,Y 580.272,Z 578.198,A -85,B 0,C 180,E1 -1963.825,E2 -1963.825} C_VEL
LIN {X 0,Y 580.317,Z 578.192,A -85,B 0,C 180,E1 -1965.983,E2 -1965.983} C_VEL
LIN {X 0,Y 580.321,Z 578.195,A -85,B 0,C 180,E1 -1968.827,E2 -1968.827} C_VEL
LIN {X 0,Y 580.328,Z 578.195,A -85,B 0,C 180,E1 -1971.644,E2 -1971.644} C_VEL
LIN {X 0,Y 580.322,Z 578.191,A -85,B 0,C 180,E1 -1974.44,E2 -1974.44} C_VEL
LIN {X 0,Y 580.34,Z 578.196,A -85,B 0,C 180,E1 -1977.223,E2 -1977.223} C_VEL
LIN {X 0,Y 580.341,Z 578.191,A -85,B 0,C 180,E1 -1980,E2 -1980} C_VEL
LIN {X 0,Y 580.34,Z 578.19,A -85,B 0,C 180,E1 -1982.776,E2 -1982.776} C_VEL
LIN {X 0,Y 580.316,Z 578.203,A -85,B 0,C 180,E1 -1985.559,E2 -1985.559} C_VEL
LIN {X 0,Y 580.327,Z 578.191,A -85,B 0,C 180,E1 -1988.356,E2 -1988.356} C_VEL
LIN {X 0,Y 580.322,Z 578.194,A -85,B 0,C 180,E1 -1991.208,E2 -1991.208} C_VEL
LIN {X 0,Y 580.303,Z 578.195,A -85,B 0,C 180,E1 -1994.339,E2 -1994.339} C_VEL
LIN {X 0,Y 580.301,Z 578.194,A -85,B 0,C 180,E1 -1996.914,E2 -1996.914} C_VEL
LIN {X 0,Y 580.297,Z 578.205,A -85,B 0,C 180,E1 -1999.822,E2 -1999.822} C_VEL
LIN {X 0,Y 580.276,Z 578.199,A -85,B 0,C 180,E1 -2001.343,E2 -2001.343} C_VEL
LIN {X 0,Y 579.578,Z 578.293,A -85,B 0,C 180,E1 -2001.922,E2 -2001.922} C_VEL
LIN {X 0,Y 576.701,Z 578.649,A -85,B 0,C 180,E1 -2002.862,E2 -2002.862} C_VEL
LIN {X 0,Y 574.307,Z 578.947,A -85,B 0,C 180,E1 -2003.618,E2 -2003.618} C_VEL
LIN {X 0,Y 573.308,Z 579.071,A -85,B 0,C 180,E1 -2004.202,E2 -2004.202} C_VEL
LIN {X 0,Y 573.241,Z 579.076,A -85,B 0,C 180,E1 -2004.4,E2 -2004.4} C_VEL
LIN {X 0,Y 573.257,Z 579.071,A -85,B 0,C 180,E1 -2006.975,E2 -2006.975} C_VEL
LIN {X 0,Y 573.243,Z 579.076,A -85,B 0,C 180,E1 -2009.49,E2 -2009.49} C_VEL
LIN {X 0,Y 573.245,Z 579.08,A -85,B 0,C 180,E1 -2012.229,E2 -2012.229} C_VEL
LIN {X 0,Y 573.241,Z 579.074,A -85,B 0,C 180,E1 -2014.774,E2 -2014.774} C_VEL
LIN {X 0,Y 573.246,Z 579.072,A -85,B 0,C 180,E1 -2017.167,E2 -2017.167} C_VEL
LIN {X 0,Y 573.242,Z 579.075,A -85,B 0,C 180,E1 -2019.607,E2 -2019.607} C_VEL
LIN {X 0,Y 573.252,Z 579.076,A -85,B 0,C 180,E1 -2022.644,E2 -2022.644} C_VEL
LIN {X 0,Y 573.23,Z 579.076,A -85,B 0,C 180,E1 -2025.667,E2 -2025.667} C_VEL
LIN {X 0,Y 573.236,Z 579.081,A -85,B 0,C 180,E1 -2028.545,E2 -2028.545} C_VEL
LIN {X 0,Y 573.241,Z 579.073,A -85,B 0,C 180,E1 -2031.3,E2 -2031.3} C_VEL
LIN {X 0,Y 573.258,Z 579.075,A -85,B 0,C 180,E1 -2034.012,E2 -2034.012} C_VEL
LIN {X 0,Y 573.279,Z 579.079,A -85,B 0,C 180,E1 -2036.519,E2 -2036.519} C_VEL
LIN {X 0,Y 573.232,Z 579.076,A -85,B 0,C 180,E1 -2039.116,E2 -2039.116} C_VEL
LIN {X 0,Y 573.259,Z 579.073,A -85,B 0,C 180,E1 -2041.969,E2 -2041.969} C_VEL
LIN {X 0,Y 573.25,Z 579.083,A -85,B 0,C 180,E1 -2044.59,E2 -2044.59} C_VEL
LIN {X 0,Y 573.234,Z 579.074,A -85,B 0,C 180,E1 -2047.663,E2 -2047.663} C_VEL
LIN {X 0,Y 573.274,Z 579.08,A -85,B 0,C 180,E1 -2050.729,E2 -2050.729} C_VEL
LIN {X 0,Y 573.255,Z 579.072,A -85,B 0,C 180,E1 -2053.622,E2 -2053.622} C_VEL
LIN {X 0,Y 573.235,Z 579.079,A -85,B 0,C 180,E1 -2056.53,E2 -2056.53} C_VEL
LIN {X 0,Y 573.259,Z 579.079,A -85,B 0,C 180,E1 -2058.745,E2 -2058.745} C_VEL
LIN {X 0,Y 573.287,Z 579.069,A -85,B 0,C 180,E1 -2061.541,E2 -2061.541} C_VEL
LIN {X 0,Y 573.294,Z 579.068,A -85,B 0,C 180,E1 -2064.372,E2 -2064.372} C_VEL
LIN {X 0,Y 573.311,Z 579.065,A -85,B 0,C 180,E1 -2067.892,E2 -2067.892} C_VEL
LIN {X 0,Y 573.327,Z 579.067,A -85,B 0,C 180,E1 -2070.702,E2 -2070.702} C_VEL
LIN {X 0,Y 573.303,Z 579.071,A -85,B 0,C 180,E1 -2072.811,E2 -2072.811} C_VEL
LIN {X 0,Y 573.296,Z 579.07,A -85,B 0,C 180,E1 -2075.628,E2 -2075.628} C_VEL
LIN {X 0,Y 573.282,Z 579.068,A -85,B 0,C 180,E1 -2078.459,E2 -2078.459} C_VEL
LIN {X 0,Y 573.269,Z 579.08,A -85,B 0,C 180,E1 -2081.312,E2 -2081.312} C_VEL
LIN {X 0,Y 573.271,Z 579.07,A -85,B 0,C 180,E1 -2084.193,E2 -2084.193} C_VEL
LIN {X 0,Y 573.256,Z 579.077,A -85,B 0,C 180,E1 -2087.111,E2 -2087.111} C_VEL
LIN {X 0,Y 573.25,Z 579.074,A -85,B 0,C 180,E1 -2090.076,E2 -2090.076} C_VEL
LIN {X 0,Y 573.229,Z 579.079,A -85,B 0,C 180,E1 -2093.099,E2 -2093.099} C_VEL
LIN {X 0,Y 573.255,Z 579.082,A -85,B 0,C 180,E1 -2095.409,E2 -2095.409} C_VEL
LIN {X 0,Y 573.322,Z 579.205,A -85,B 0,C 180,E1 -2096.664,E2 -2096.664} C_VEL
LIN {X 0,Y 573.344,Z 592.483,A -85,B 0,C 180,E1 -2099.159,E2 -2099.159} C_VEL
LIN {X 0,Y 573.232,Z 603.61,A -85,B 0,C 180,E1 -2101.223,E2 -2101.223} C_VEL
LIN {X 0,Y 574.076,Z 609.426,A -85,B 0,C 180,E1 -2101.326,E2 -2101.326} C_VEL
LIN {X 0,Y 573.863,Z 710.806,A -85,B 0,C 180,E1 -2102.618,E2 -2102.618} C_VEL
LIN {X 0,Y 573.768,Z 724.446,A -85,B 0,C 180,E1 -2102.95,E2 -2102.95} C_VEL
LIN {X 0,Y 573.683,Z 736.909,A -85,B 0,C 180,E1 -2103.401,E2 -2103.401} C_VEL
LIN {X 0,Y 573.57,Z 747.497,A -85,B 0,C 180,E1 -2103.91,E2 -2103.91} C_VEL
LIN {X 0,Y 573.443,Z 758.377,A -85,B 0,C 180,E1 -2104.573,E2 -2104.573} C_VEL
LIN {X 0,Y 573.338,Z 769.143,A -85,B 0,C 180,E1 -2105.393,E2 -2105.393} C_VEL
LIN {X 0,Y 573.246,Z 778.464,A -85,B 0,C 180,E1 -2106.266,E2 -2106.266} C_VEL
LIN {X 0,Y 573.159,Z 787.226,A -85,B 0,C 180,E1 -2107.279,E2 -2107.279} C_VEL
LIN {X 0,Y 573.101,Z 794.365,A -85,B 0,C 180,E1 -2108.295,E2 -2108.295} C_VEL
LIN {X 0,Y 573.048,Z 800.65,A -85,B 0,C 180,E1 -2109.408,E2 -2109.408} C_VEL
LIN {X 0,Y 573.003,Z 805.66,A -85,B 0,C 180,E1 -2110.545,E2 -2110.545} C_VEL
LIN {X 0,Y 573.001,Z 810.142,A -85,B 0,C 180,E1 -2111.967,E2 -2111.967} C_VEL
LIN {X 0,Y 572.966,Z 811.597,A -85,B 0,C 180,E1 -2112.612,E2 -2112.612} C_VEL
LIN {X 0,Y 572.919,Z 813.181,A -85,B 0,C 180,E1 -2113.635,E2 -2113.635} C_VEL
LIN {X 0,Y 572.926,Z 813.917,A -85,B 0,C 180,E1 -2114.645,E2 -2114.645} C_VEL
LIN {X 0,Y 572.93,Z 813.857,A -85,B 0,C 180,E1 -2115.637,E2 -2115.637} C_VEL
LIN {X 0,Y 572.927,Z 813.003,A -85,B 0,C 180,E1 -2116.612,E2 -2116.612} C_VEL
LIN {X 0,Y 572.993,Z 811.392,A -85,B 0,C 180,E1 -2117.578,E2 -2117.578} C_VEL
LIN {X 0,Y 572.995,Z 809.07,A -85,B 0,C 180,E1 -2118.523,E2 -2118.523} C_VEL
LIN {X 0,Y 573.003,Z 805.835,A -85,B 0,C 180,E1 -2119.502,E2 -2119.502} C_VEL
LIN {X 0,Y 573.047,Z 801.113,A -85,B 0,C 180,E1 -2120.591,E2 -2120.591} C_VEL
LIN {X 0,Y 573.092,Z 794.932,A -85,B 0,C 180,E1 -2121.705,E2 -2121.705} C_VEL
LIN {X 0,Y 573.163,Z 786.974,A -85,B 0,C 180,E1 -2122.844,E2 -2122.844} C_VEL
LIN {X 0,Y 573.245,Z 778.283,A -85,B 0,C 180,E1 -2123.843,E2 -2123.843} C_VEL
LIN {X 0,Y 573.373,Z 767.626,A -85,B 0,C 180,E1 -2124.824,E2 -2124.824} C_VEL
LIN {X 0,Y 573.463,Z 757.17,A -85,B 0,C 180,E1 -2125.6,E2 -2125.6} C_VEL
LIN {X 0,Y 573.586,Z 745.011,A -85,B 0,C 180,E1 -2126.308,E2 -2126.308} C_VEL
LIN {X 0,Y 573.751,Z 732.503,A -85,B 0,C 180,E1 -2126.865,E2 -2126.865} C_VEL
LIN {X 0,Y 573.812,Z 719.698,A -85,B 0,C 180,E1 -2127.274,E2 -2127.274} C_VEL
LIN {X 0,Y 573.877,Z 706.588,A -85,B 0,C 180,E1 -2127.541,E2 -2127.541} C_VEL
LIN {X 0,Y 574.034,Z 608.738,A -85,B 0,C 180,E1 -2128.774,E2 -2128.774} C_VEL
LIN {X 0,Y 573.248,Z 603.537,A -85,B 0,C 180,E1 -2128.88,E2 -2128.88} C_VEL
LIN {X 0,Y 573.357,Z 589.742,A -85,B 0,C 180,E1 -2131.443,E2 -2131.443} C_VEL
LIN {X 0,Y 573.29,Z 579.161,A -85,B 0,C 180,E1 -2133.435,E2 -2133.435} C_VEL
LIN {X 0,Y 573.224,Z 579.081,A -85,B 0,C 180,E1 -2136.135,E2 -2136.135} C_VEL
LIN {X 0,Y 573.251,Z 579.075,A -85,B 0,C 180,E1 -2139.174,E2 -2139.174} C_VEL
LIN {X 0,Y 573.231,Z 579.076,A -85,B 0,C 180,E1 -2141.412,E2 -2141.412} C_VEL
LIN {X 0,Y 573.249,Z 579.073,A -85,B 0,C 180,E1 -2143.622,E2 -2143.622} C_VEL
LIN {X 0,Y 573.233,Z 579.083,A -85,B 0,C 180,E1 -2146.53,E2 -2146.53} C_VEL
LIN {X 0,Y 573.267,Z 579.072,A -85,B 0,C 180,E1 -2149.404,E2 -2149.404} C_VEL
LIN {X 0,Y 573.282,Z 579.071,A -85,B 0,C 180,E1 -2152.25,E2 -2152.25} C_VEL
LIN {X 0,Y 573.31,Z 579.071,A -85,B 0,C 180,E1 -2155.078,E2 -2155.078} C_VEL
LIN {X 0,Y 573.3,Z 579.066,A -85,B 0,C 180,E1 -2157.893,E2 -2157.893} C_VEL
LIN {X 0,Y 573.329,Z 579.07,A -85,B 0,C 180,E1 -2160.703,E2 -2160.703} C_VEL
LIN {X 0,Y 573.236,Z 579.075,A -85,B 0,C 180,E1 -2163.515,E2 -2163.515} C_VEL
LIN {X 0,Y 573.293,Z 579.068,A -85,B 0,C 180,E1 -2165.629,E2 -2165.629} C_VEL
LIN {X 0,Y 573.3,Z 579.069,A -85,B 0,C 180,E1 -2168.46,E2 -2168.46} C_VEL
LIN {X 0,Y 573.289,Z 579.073,A -85,B 0,C 180,E1 -2171.312,E2 -2171.312} C_VEL
LIN {X 0,Y 573.271,Z 579.071,A -85,B 0,C 180,E1 -2174.425,E2 -2174.425} C_VEL
LIN {X 0,Y 573.251,Z 579.083,A -85,B 0,C 180,E1 -2177.112,E2 -2177.112} C_VEL
LIN {X 0,Y 573.249,Z 579.072,A -85,B 0,C 180,E1 -2180.077,E2 -2180.077} C_VEL
LIN {X 0,Y 573.23,Z 579.075,A -85,B 0,C 180,E1 -2182.338,E2 -2182.338} C_VEL
LIN {X 0,Y 573.25,Z 579.079,A -85,B 0,C 180,E1 -2185.411,E2 -2185.411} C_VEL
LIN {X 0,Y 573.256,Z 579.071,A -85,B 0,C 180,E1 -2188.032,E2 -2188.032} C_VEL
LIN {X 0,Y 573.238,Z 579.077,A -85,B 0,C 180,E1 -2190.886,E2 -2190.886} C_VEL
LIN {X 0,Y 573.282,Z 579.075,A -85,B 0,C 180,E1 -2193.529,E2 -2193.529} C_VEL
LIN {X 0,Y 573.255,Z 579.073,A -85,B 0,C 180,E1 -2196.049,E2 -2196.049} C_VEL
LIN {X 0,Y 573.246,Z 579.073,A -85,B 0,C 180,E1 -2198.702,E2 -2198.702} C_VEL
LIN {X 0,Y 573.25,Z 579.08,A -85,B 0,C 180,E1 -2201.597,E2 -2201.597} C_VEL
LIN {X 0,Y 573.235,Z 579.075,A -85,B 0,C 180,E1 -2204.334,E2 -2204.334} C_VEL
LIN {X 0,Y 573.237,Z 579.082,A -85,B 0,C 180,E1 -2207.359,E2 -2207.359} C_VEL
LIN {X 0,Y 573.245,Z 579.073,A -85,B 0,C 180,E1 -2210.394,E2 -2210.394} C_VEL
LIN {X 0,Y 573.254,Z 579.075,A -85,B 0,C 180,E1 -2213.079,E2 -2213.079} C_VEL
LIN {X 0,Y 573.273,Z 579.08,A -85,B 0,C 180,E1 -2215.673,E2 -2215.673} C_VEL
LIN {X 0,Y 573.242,Z 579.076,A -85,B 0,C 180,E1 -2218.185,E2 -2218.185} C_VEL
LIN {X 0,Y 573.265,Z 579.071,A -85,B 0,C 180,E1 -2220.635,E2 -2220.635} C_VEL
LIN {X 0,Y 573.251,Z 579.075,A -85,B 0,C 180,E1 -2223.025,E2 -2223.025} C_VEL
LIN {X 0,Y 573.265,Z 579.145,A -85,B 0,C 180,E1 -2226.041,E2 -2226.041} C_VEL
LIN {X 0,Y 574.052,Z 583.25,A -85,B 0,C 180,E1 -2226.666,E2 -2226.666} C_VEL
LIN {X 0,Y 573.953,Z 598.72,A -85,B 0,C 180,E1 -2228.867,E2 -2228.867} C_VEL
LIN {X 0,Y 573.706,Z 619.698,A -85,B 0,C 180,E1 -2231.798,E2 -2231.798} C_VEL
LIN {X 0,Y 573.502,Z 639.641,A -85,B 0,C 180,E1 -2234.542,E2 -2234.542} C_VEL
LIN {X 0,Y 573.413,Z 651.524,A -85,B 0,C 180,E1 -2236.161,E2 -2236.161} C_VEL
LIN {X 0,Y 574.101,Z 657.536,A -85,B 0,C 180,E1 -2236.257,E2 -2236.257} C_VEL
LIN {X 0,Y 573.903,Z 759.962,A -85,B 0,C 180,E1 -2237.558,E2 -2237.558} C_VEL
LIN {X 0,Y 573.801,Z 772.468,A -85,B 0,C 180,E1 -2237.848,E2 -2237.848} C_VEL
LIN {X 0,Y 573.703,Z 785.38,A -85,B 0,C 180,E1 -2238.294,E2 -2238.294} C_VEL
LIN {X 0,Y 573.575,Z 797.735,A -85,B 0,C 180,E1 -2238.879,E2 -2238.879} C_VEL
LIN {X 0,Y 573.44,Z 809.207,A -85,B 0,C 180,E1 -2239.585,E2 -2239.585} C_VEL
LIN {X 0,Y 573.327,Z 819.602,A -85,B 0,C 180,E1 -2240.386,E2 -2240.386} C_VEL
LIN {X 0,Y 573.241,Z 828.115,A -85,B 0,C 180,E1 -2241.185,E2 -2241.185} C_VEL
LIN {X 0,Y 573.161,Z 835.962,A -85,B 0,C 180,E1 -2242.071,E2 -2242.071} C_VEL
LIN {X 0,Y 573.073,Z 843.955,A -85,B 0,C 180,E1 -2243.186,E2 -2243.186} C_VEL
LIN {X 0,Y 573.07,Z 850.681,A -85,B 0,C 180,E1 -2244.37,E2 -2244.37} C_VEL
LIN {X 0,Y 573.029,Z 855.372,A -85,B 0,C 180,E1 -2245.428,E2 -2245.428} C_VEL
LIN {X 0,Y 573.023,Z 858.957,A -85,B 0,C 180,E1 -2246.484,E2 -2246.484} C_VEL
LIN {X 0,Y 572.959,Z 860.809,A -85,B 0,C 180,E1 -2247.188,E2 -2247.188} C_VEL
LIN {X 0,Y 572.937,Z 862.199,A -85,B 0,C 180,E1 -2247.891,E2 -2247.891} C_VEL
LIN {X 0,Y 572.941,Z 863.785,A -85,B 0,C 180,E1 -2249.297,E2 -2249.297} C_VEL
LIN {X 0,Y 572.938,Z 864,A -85,B 0,C 180,E1 -2250,E2 -2250} C_VEL
LIN {X 0,Y 572.946,Z 863.186,A -85,B 0,C 180,E1 -2251.406,E2 -2251.406} C_VEL
LIN {X 0,Y 572.937,Z 862.2,A -85,B 0,C 180,E1 -2252.109,E2 -2252.109} C_VEL
LIN {X 0,Y 572.959,Z 860.81,A -85,B 0,C 180,E1 -2252.812,E2 -2252.812} C_VEL
LIN {X 0,Y 573.015,Z 857.896,A -85,B 0,C 180,E1 -2253.868,E2 -2253.868} C_VEL
LIN {X 0,Y 572.963,Z 853.95,A -85,B 0,C 180,E1 -2254.925,E2 -2254.925} C_VEL
LIN {X 0,Y 573.064,Z 847.878,A -85,B 0,C 180,E1 -2256.16,E2 -2256.16} C_VEL
LIN {X 0,Y 573.119,Z 841.238,A -85,B 0,C 180,E1 -2257.221,E2 -2257.221} C_VEL
LIN {X 0,Y 573.201,Z 832.992,A -85,B 0,C 180,E1 -2258.283,E2 -2258.283} C_VEL
LIN {X 0,Y 573.286,Z 824.54,A -85,B 0,C 180,E1 -2259.17,E2 -2259.17} C_VEL
LIN {X 0,Y 573.423,Z 814.1,A -85,B 0,C 180,E1 -2260.058,E2 -2260.058} C_VEL
LIN {X 0,Y 573.549,Z 802.359,A -85,B 0,C 180,E1 -2260.857,E2 -2260.857} C_VEL
LIN {X 0,Y 573.653,Z 791.287,A -85,B 0,C 180,E1 -2261.447,E2 -2261.447} C_VEL
LIN {X 0,Y 573.775,Z 778.183,A -85,B 0,C 180,E1 -2261.973,E2 -2261.973} C_VEL
LIN {X 0,Y 573.824,Z 765.533,A -85,B 0,C 180,E1 -2262.331,E2 -2262.331} C_VEL
LIN {X 0,Y 573.915,Z 752.335,A -85,B 0,C 180,E1 -2262.554,E2 -2262.554} C_VEL
LIN {X 0,Y 573.991,Z 655.301,A -85,B 0,C 180,E1 -2263.773,E2 -2263.773} C_VEL
LIN {X 0,Y 573.419,Z 651.441,A -85,B 0,C 180,E1 -2263.85,E2 -2263.85} C_VEL
LIN {X 0,Y 573.623,Z 628.373,A -85,B 0,C 180,E1 -2267.004,E2 -2267.004} C_VEL
LIN {X 0,Y 573.866,Z 606.402,A -85,B 0,C 180,E1 -2270.054,E2 -2270.054} C_VEL
LIN {X 0,Y 574.141,Z 586.458,A -85,B 0,C 180,E1 -2272.87,E2 -2272.87} C_VEL
LIN {X 0,Y 573.833,Z 581.934,A -85,B 0,C 180,E1 -2273.532,E2 -2273.532} C_VEL
LIN {X 0,Y 573.254,Z 579.08,A -85,B 0,C 180,E1 -2274.008,E2 -2274.008} C_VEL
LIN {X 0,Y 573.251,Z 579.075,A -85,B 0,C 180,E1 -2276.975,E2 -2276.975} C_VEL
LIN {X 0,Y 573.247,Z 579.074,A -85,B 0,C 180,E1 -2279.488,E2 -2279.488} C_VEL
LIN {X 0,Y 573.255,Z 579.078,A -85,B 0,C 180,E1 -2282.644,E2 -2282.644} C_VEL
LIN {X 0,Y 573.267,Z 579.071,A -85,B 0,C 180,E1 -2285.183,E2 -2285.183} C_VEL
LIN {X 0,Y 573.233,Z 579.075,A -85,B 0,C 180,E1 -2287.807,E2 -2287.807} C_VEL
LIN {X 0,Y 573.267,Z 579.08,A -85,B 0,C 180,E1 -2290.527,E2 -2290.527} C_VEL
LIN {X 0,Y 573.24,Z 579.073,A -85,B 0,C 180,E1 -2293.668,E2 -2293.668} C_VEL
LIN {X 0,Y 573.243,Z 579.083,A -85,B 0,C 180,E1 -2296.641,E2 -2296.641} C_VEL
LIN {X 0,Y 573.269,Z 579.07,A -85,B 0,C 180,E1 -2299.477,E2 -2299.477} C_VEL
LIN {X 0,Y 573.232,Z 579.076,A -85,B 0,C 180,E1 -2302.192,E2 -2302.192} C_VEL
LIN {X 0,Y 573.261,Z 579.082,A -85,B 0,C 180,E1 -2304.816,E2 -2304.816} C_VEL
LIN {X 0,Y 573.249,Z 579.075,A -85,B 0,C 180,E1 -2307.354,E2 -2307.354} C_VEL
